(* CODESYS project rscommcommon.library
   Company: ESO
   Description: Common library for all rsComm projects.
   Version: 0.2.0.2
   Placeholder: ESO LDC Comm Common Library
   Title: ESO LDC Comm Common Library

Project tree, tasks and I/O mapping:
  libraries: Tc2_Standard, * (Beckhoff Automation GmbH); Tc2_System, * (Beckhoff Automation GmbH); Tc2_Utilities, * (Beckhoff Automation GmbH); Tc3_Module, * (Beckhoff Automation GmbH)
  DUTs/
    Enumerated/
      Comm/
        data type E_MODBUS_CMD_TYPE
        data type E_RS_BASE_READ_TYPE
        data type E_RS_COMM_CMD
        data type E_RS_COMM_ERROR
        data type E_RS_COMM_STATE
        data type E_RS_COMM_STATUS
        data type E_RS_COMMAND
        data type E_RS_RPC_ERROR
      Devices/
        data type E_LAKESHORE_CMD_TYPE
        data type E_LAKESHORE_ERROR
        data type E_RS_BASE_STATE
        data type E_RS_BASE_SUBSTATE
        data type E_SM_ERROR
        data type E_SM_EVENT
        data type E_SM_STATUS
    Structures/
      Comm/
        data type T_READING_LREAL
        data type T_RS_COMM_CFG
        data type T_RS_COMM_CTRL
        data type T_RS_COMM_INFO
        data type T_RS_COMM_STAT
      Devices/
        data type T_LAKESHORE_CFG
        data type T_LAKESHORE_COMMAND
        data type T_LAKESHORE_CTRL
        data type T_LAKESHORE_INFO
        data type T_LAKESHORE_STAT
        data type T_RS_BASE_CFG
        data type T_RS_BASE_CTRL
        data type T_RS_BASE_STAT
  GVLs/
  lib/
  POUs/
    function block FB_LAKESHORE_BASE [ST]: ActionInitExecute, ActivityInitializing, ActivityMonitoring, ActivityMonitoringUser, CheckForEvents, M_CheckCmdIndex, M_Configure, M_GetCommand, M_GetCommInitialised, M_GetCommStatus, M_GetCouplerState, M_RampDisable, M_RampEnable, M_ReadFromReply, M_UpdateStatus, ProcessEvents
    function block FB_RS_BASE [ST]: ActionDisableExecute, ActionEnableExecute, ActionErrExecute, ActionInitExecute, ActionResetExecute, ActionStopExecute, ActionUnexpExecute, ActivityInitializing, ActivityMonitoring, ActivityMonitoringUser, CheckForEvents, M_Configure, M_GetCouplerState, M_GetRpcErrorText, M_ReadSensors, M_SetLastGoodSubstate, M_SetRpcStatus, ProcessEvents, RPC_Disable, RPC_Enable, RPC_Init, RPC_Reset, RPC_Stop, SetAction, SetEvent, SetLastCommand, SetState, SetStatus
    function block FB_SIM_MODBUS_COMM_BASE [ST]: M_ActivityDo, M_ByteSwap_INT_TO_BYTES, M_ByteSwap_INT_TO_STRING, M_ByteSwap_REAL_TO_BYTES, M_ByteSwap_REAL_TO_STRING, M_ByteSwap_UINT_TO_BYTES, M_ByteSwapINT, M_ByteSwapREAL, M_GenerateRandom_INT, M_GenerateRandom_REAL, M_GetSimReply, M_InsertBytes_INT, M_InsertBytes_REAL
    function block FB_SIM_MODBUS_COMM_JUMO [ST]: M_GetSimReply
    function block FB_SIM_RS_COMM_BASE [ST]: M_ActivityDo, M_GenerateRandom_LREAL, M_Get_INT_TO_STRING, M_Get_LREAL_TO_STRING, M_GetRandom_LREAL_TO_STRING, M_GetSimReply
    function block FB_SIM_RS_COMM_DUMMY [ST]: M_ActivityDo, M_GetSimReply
    function block FB_SIM_RS_COMM_LAKESHORE [ST]: M_ActivityDo, M_GetSimReply
    program MAIN [ST]
  VISUs/
*)

// DUTs/Enumerated/Comm/E_MODBUS_CMD_TYPE
{attribute 'qualified_only'}
{attribute 'strict'}
TYPE E_MODBUS_CMD_TYPE :
(
	READ	:=	0,
	WRITE	:=	1
);
END_TYPE

// DUTs/Enumerated/Comm/E_RS_BASE_READ_TYPE
{attribute 'qualified_only'}
{attribute 'strict'}
TYPE E_RS_BASE_READ_TYPE :
(
	SINGLE			:= 0,
	SINGLE_USER,
	PERIODIC,
	PERIODIC_USER
);
END_TYPE

// DUTs/Enumerated/Comm/E_RS_COMM_CMD
{attribute 'qualified_only'}
////{xxxattribute 'strict'}
TYPE E_RS_COMM_CMD :
(
	NONE		:=	0,
	INIT		:=	1,
	SEND		:=	2,
	DISCONNECT	:=	3
);
END_TYPE

// DUTs/Enumerated/Comm/E_RS_COMM_ERROR
{attribute 'qualified_only'}
//{attribute 'strict'}
TYPE E_RS_COMM_ERROR :
(
	OK				:= 0,
	NOT_IN_OP_STATE,
	NOT_INIT,
	TIMEOUT,
	LISTEN,
	ACCEPT,
	SEND,
	RECEIVE,
	WRONG_STATE,
	NOT_IDLE,
	CONNECT,
	DISCONNECT
);
END_TYPE

// DUTs/Enumerated/Comm/E_RS_COMM_STATE
{attribute 'qualified_only'}
{attribute 'strict'}
TYPE E_RS_COMM_STATE :
(
	NOT_INIT			:= 0,
	IDLE				:= 1,
	CONNECT				:= 2,
	RESET				:= 3,
	PREPARE_SEND		:= 5,
	SEND				:= 10,
	RECEIVE				:= 15,
	WAIT				:= 20,
	CLEAR_BUFFER		:= 40,
	WAIT_AFTER_SEND		:= 55,
	DISCONNECT			:= 60,

	ERROR				:= 100
);
END_TYPE

// DUTs/Enumerated/Comm/E_RS_COMM_STATUS
{attribute 'qualified_only'}
////{xxxattribute 'strict'}
TYPE E_RS_COMM_STATUS :
(
	NOT_INIT	:= -1,
	IDLE		:= 0,
	BUSY		:= 1,
	ERROR		:= 2
);
END_TYPE

// DUTs/Enumerated/Comm/E_RS_COMMAND
{attribute 'qualified_only'}
{attribute 'strict'}
TYPE E_RS_COMMAND :
(
	NONE	:= 0,
	
	RESET,
	INIT,
	STOP,
	ENABLE,
	DISABLE,
	
	READ,
	READ_USER,
	MONITOR,
	MONITOR_USER,
	STOPMON,
	
	CTRL_CMD
	
);
END_TYPE

// DUTs/Enumerated/Comm/E_RS_RPC_ERROR
{attribute 'qualified_only'}
//{attribute 'strict'}
TYPE E_RS_RPC_ERROR :
(
	OK					:= 0,
	NOT_OP				:= -1,			
	NOT_NOTOP_READY		:= -2,			
	NOT_NOTOP_NOTREADY	:= -3,			
	LOCAL				:= -4			
);
END_TYPE

// DUTs/Enumerated/Devices/E_LAKESHORE_CMD_TYPE
{attribute 'qualified_only'}
{attribute 'strict'}
TYPE E_LAKESHORE_CMD_TYPE :
(
	INIT := 0,
	READ,
	CTRL
);
END_TYPE

// DUTs/Enumerated/Devices/E_LAKESHORE_ERROR
TYPE E_LAKESHORE_ERROR :
(
	OK				:= 16#0000,
	NOT_IN_OP_STATE	:= 16#0001,
	NOT_INIT		:= 16#0002,
	TIMEOUT			:= 16#0004,
	COMM			:= 16#0008,
	WRONG_STATE		:= 16#0010,
	NOT_IDLE		:= 16#0020
);
END_TYPE

// DUTs/Enumerated/Devices/E_RS_BASE_STATE
{attribute 'qualified_only'}
//{attribute 'strict'}
TYPE E_RS_BASE_STATE :
(
	NONE	:= 0,
	NOTOP,
	OP
);
END_TYPE

// DUTs/Enumerated/Devices/E_RS_BASE_SUBSTATE
// Substates MUST match definitions in the WS driver that can be found in
// ICS/ifw/fcf/devmgr/devices/src/include/devmgr/devices/sensorConfig.hpp
// Never change them without consulting the team.
{attribute 'qualified_only'}
//{attribute 'strict'}
TYPE E_RS_BASE_SUBSTATE :
(
	NONE				:= 0,
	
	NOTOP_NOTREADY		:= 100,
	NOTOP_READY			:= 101,
	NOTOP_INITIALIZING	:= 102,
	NOTOP_ERROR			:= 199,
	
	OP_MONITORING   	:= 200,
	OP_IDLE         	:= 201,
	OP_MONITORING_USER	:= 202,
	OP_ERROR         	:= 299
);
END_TYPE

// DUTs/Enumerated/Devices/E_SM_ERROR
{attribute 'qualified_only'}
//{attribute 'strict'}
TYPE E_SM_ERROR :
(
	OK					:= 0,
	HW_NOT_OP,			
	WRONG_CMD,			
	INIT_FAILURE,		

	NOT_INITIALISED		:= 90,
	ZERO_POINTER		:= 100	// Simulator error
);
END_TYPE

// DUTs/Enumerated/Devices/E_SM_EVENT
TYPE E_SM_EVENT :
(
	NONE	:= 0,
	
	(* events corresponding to commands *)
	RESET,
	INIT,
	STOP,
	ENABLE,
	DISABLE,
	
	READ,
	READ_USER,
	MONITOR,
	MONITOR_USER,
	STOPMON,
	CTRL_CMD,
	
	(* 
		Events corresponding to internal events 
	*)
	INITDONE,
	READDONE,
	
	
	(* events mapped to HW signals *)
	HWOK,
	COMMOK,
	ERRCOMM,
	ERRHW,
	ERRINIT
	
);
END_TYPE

// DUTs/Enumerated/Devices/E_SM_STATUS
TYPE E_SM_STATUS :
(
	OK		:= 0,
	ERROR
);
END_TYPE

// DUTs/Structures/Comm/T_READING_LREAL
TYPE T_READING_LREAL :
STRUCT
	lrValue:	LREAL; 	// LREAL (DOUBLE)
END_STRUCT
END_TYPE

// DUTs/Structures/Comm/T_RS_COMM_CFG
TYPE T_RS_COMM_CFG :
STRUCT

	sCmdSuffix:		STRING(16) := '$0D$0A';	(* Terminator for command *)
	sReplySuffix:	STRING(16) := '$0D$0A';	(* Terminator for reply *)

	nTimeout:		DINT := 3000;			(* Timeout on command reply. ALWAYS use ms for time !!! *)

END_STRUCT
END_TYPE

// DUTs/Structures/Comm/T_RS_COMM_CTRL
TYPE T_RS_COMM_CTRL :
STRUCT
	(* CTRL *)
	nCommand:		E_RS_COMM_CMD := E_RS_COMM_CMD.NONE;	(* Command Number, e.g. to INIT or SEND a command *)
	bExecute:		BOOL;						(* Setting to TRUE activates command *)

	sCmd:			STRING := '';				(* Command to be sent, e.g. '*IDN?' to get Lakeshore ID*)

	bHasReply:		BOOL;						(* If TRUE, there is a reply to the command *)

	nNumReplies:	DINT := 1;	(* Number of replies, i.e. number of cfg.sReplySuffix strings expected in the reply *)

END_STRUCT
END_TYPE

// DUTs/Structures/Comm/T_RS_COMM_INFO
TYPE T_RS_COMM_INFO :
STRUCT
(*
	Driver Information

	Change LOG:
	0.1 2018-02-07	- Copy of VLT RS_Comm_TC3 project @306329.
*)

	sDate:			STRING(32)	:= '2018-02-06';
	sDescription:	STRING(80) 	:= 'Serial Port Communication Drivers';
	sName:			STRING(64)	:= 'FB_RS_COMM';
	sPlatform:		STRING(32)	:= 'CoDeSys';
	sSynopsis:		STRING(64)	:= 'Serial Port Communication Drivers';
	nVersionMajor:	DINT		:= 0;
	nVersionMinor:	DINT		:= 1;


END_STRUCT
END_TYPE

// DUTs/Structures/Comm/T_RS_COMM_STAT
TYPE T_RS_COMM_STAT :
STRUCT
	(* STAT *)
	bInitialised:		BOOL := FALSE;		(* Flag if device is initialised *)
	bSimulation:		BOOL := FALSE;		(* Device simulated *)
	bConnected:			BOOL := FALSE;		(* Established connection status *)


	nLastCommand:		E_RS_COMM_CMD 		:= E_RS_COMM_CMD.NONE;
	nErrorCode:			E_RS_COMM_ERROR 	:= E_RS_COMM_ERROR.OK;
	nStatus: 			E_RS_COMM_STATUS	:= E_RS_COMM_STATUS.NOT_INIT; (* See E_RS_COMM_STATUS definitions *)

	sErrorText: 		STRING 	:= 'OK';
	sStatus:			STRING	:= '';			(* Status description *)

	sReply:				STRING(255);			(* Last  Reply from the device *)

END_STRUCT
END_TYPE

// DUTs/Structures/Devices/T_LAKESHORE_CFG
TYPE T_LAKESHORE_CFG EXTENDS T_RS_BASE_CFG:
STRUCT
	cmdList_Init:	ARRAY [1..8]	OF T_LAKESHORE_COMMAND;	// List of INIT commands
	cmdList_Read:	ARRAY [1..16] 	OF T_LAKESHORE_COMMAND;	// List of READ commands

	nModel:			DINT := 336;		// Supported models: 218, 224, 340 and 336.

END_STRUCT
END_TYPE

// DUTs/Structures/Devices/T_LAKESHORE_COMMAND
TYPE T_LAKESHORE_COMMAND :
STRUCT
	cmd:		STRING := '';	(* Command to send *)
	nReplies:	DINT;   		(* Number of replies, i.e. reply terminators *)
	nValues:	DINT;   		(* Number of returned numbers (values) in the reply *)
	offset:		DINT;			(* Offset in data array where to write the first value *)
END_STRUCT
END_TYPE

// DUTs/Structures/Devices/T_LAKESHORE_CTRL
TYPE T_LAKESHORE_CTRL EXTENDS T_RS_BASE_CTRL:
STRUCT
	sCmdUser:	T_LAKESHORE_COMMAND := (cmd := '*IDN?', nReplies := 1, nValues := 1, offset := 0);

	cmdList_Ctrl:	ARRAY [1..8] OF T_LAKESHORE_COMMAND;	// List of up to 8 Ctrl Commands (no '?')

	
	nPID_A_P:			UINT;		// P controller value
	nPID_A_I:			UINT;		// I controller value
	nPID_A_D:			UINT;		// D controller value
	nHeaterRange:		UINT;		// Resistance power range
	lrCtrlRamp:			LREAL;		// Delta-T Kelvin per minutes
	lrSetpoint_A:		LREAL;		// Setpoint [K]

END_STRUCT
END_TYPE

// DUTs/Structures/Devices/T_LAKESHORE_INFO
TYPE T_LAKESHORE_INFO :
STRUCT
(*
	Driver Information

	Change LOG:
	1.0	12/02/2014	- Ported from TC2.
	1.1	13/02/2014	- Addition of input parameters for Model and readout period.
	1.2	18/02/2014	- STATUS_LAKESHORE_ERROR := 1, to match IODev ICD.
					- Disabled OPC UA for comm instance of FB_RS_COMM.
	1.3 15/10/2014	- References Newest version always
					- Removed Tc2_OpcUa from References
	2.0 2016-08-10	- OPC UA notation with TMC Files
*)
	sDate:			STRING(16)	:= '2016-08-10';
	sDescription:	STRING(32) 	:= 'Lakeshore controller';
	sName:			STRING(16)	:= 'FB_LAKESHORE';
	sPlatform:		STRING(16)	:= 'CoDeSys';
	sSynopsis:		STRING(48)	:= 'EtherCAT PLC Lakeshore controller';
	nVersionMajor:	DINT		:= 2;
	nVersionMinor:	DINT		:= 0;

END_STRUCT
END_TYPE

// DUTs/Structures/Devices/T_LAKESHORE_STAT
TYPE T_LAKESHORE_STAT EXTENDS T_RS_BASE_STAT:
STRUCT

	nRetries:			UDINT := 0;			// Total number of retries in case of communication problems
	
	lrArrReadings:		ARRAY [0..31] OF	T_READING_LREAL;	// Array of readings

	sReply:				STRING(255); 		(* Last Lakeshore Reply to predefined commands*)
	sReplyUser:			STRING(255); 		(* Last Lakeshore Reply to USER command *)

	// Lakeshore readings
	lrKRDG_A:		LREAL;	// Temperature A [K]
	lrKRDG_B:		LREAL;	// Temperature B [K]
	lrCRDG_A:		LREAL;	// Temperature A [C]
	lrCRDG_B:		LREAL;	// Temperature B [C]

	nPID_P:			UINT;	// PID parameter P
	nPID_I:			UINT;	// PID parameter I
	nPID_D:			UINT;	// PID parameter D
	bRAMP_On:		BOOL;	// RAMP 1 On/Off state
	lrRAMP_Rate:	LREAL;	// RAMP rate
	lrSETP:			LREAL;	// Actual Setpoint [K]
	lrSETP_Target:	LREAL;	// Target Setpoint [K]
	lrHTR:			LREAL;	// Heater output [%]
	nRANGE:			UINT;	// Heater range

	nPID2_P:		UINT;	// PID2 parameter P
	nPID2_I:		UINT;	// PID2 parameter I
	nPID2_D:		UINT;	// PID2 parameter D
	bRAMP2_On:		BOOL;	// RAMP 2 On/Off state
	lrRAMP2_Rate:	LREAL;	// RAMP rate
	lrSETP2:		LREAL;	// Actual Setpoint 2 [K]
	lrSETP2_Target:	LREAL;	// Target Setpoint 2 [K]
	lrHTR2:			LREAL;	// Heater2 output [%]
	nRANGE2:		UINT;	// Heater2 range

	lrAOUT1:		LREAL;	// Analog Output 1
	lrAOUT2:		LREAL;	// Analog Output 2
	lrAOUT3:		LREAL;	// Analog Output 3
	lrAOUT4:		LREAL;	// Analog Output 4
	
	
END_STRUCT
END_TYPE

// DUTs/Structures/Devices/T_RS_BASE_CFG
TYPE T_RS_BASE_CFG :
STRUCT
	tDelay_Periodic:	TIME := T#5000MS;	// Delay between sets of PERIODIC reads.
	tDelay_Init:		TIME := T#500MS;	// Delay between INIT commands
	tDelay_Ctrl:		TIME := T#100MS;	// Delay between CTRL commands
	bAutoMonitor:		BOOL := TRUE;		// If true, it starts PERIODIC reads (monitoring) after INIT
END_STRUCT
END_TYPE

// DUTs/Structures/Devices/T_RS_BASE_CTRL
TYPE T_RS_BASE_CTRL :
STRUCT
	(* CTRL *)
// DPO	nCommand:	E_RS_COMM_CMD := E_RS_COMM_CMD.NONE;
	nCommand:	E_RS_COMMAND := E_RS_COMMAND.NONE;
	bExecute:	BOOL;
	
	// User parameters used with E_RS_COMMAND.CTRL_CMD,
	// when device specific commands have to be defined.
	// Command can be specified with a combination of parameters.
	// For example:
	//    cmd := E_RS_COMMAND.CTRL_CMD & nPar1 := 1  ==> cmd = 'start pulse'
	//    cmd := E_RS_COMMAND.CTRL_CMD & nPar1 := 2  ==> cmd = 'stop pulse'
	//    cmd := E_RS_COMMAND.CTRL_CMD & nPar1 := 3  ==> cmd = 'reload'
	nPar1:		DINT;
	nPar2:		DINT;
	nPar3:		DINT;
	
	lrPar1:		LREAL;
	lrPar2:		LREAL;
	lrPar3:		LREAL;
END_STRUCT
END_TYPE

// DUTs/Structures/Devices/T_RS_BASE_STAT
TYPE T_RS_BASE_STAT :
STRUCT
	bInitialised:	BOOL 	:= FALSE;		// Flag if device is initialised
	bConfigured:	BOOL 	:= FALSE;		// Flag if device is configured
	bLocal:			BOOL	:= FALSE;		// Device operated from PLC GUI
	bSimulation:	BOOL	:= FALSE;		// Device simulated
	bAutoStarted:	BOOL	:= FALSE;		// Device has already automatically got to OP state
	bActive:		BOOL	:= FALSE;		// Device has passed first 100 cycles
	bCmdActive:		BOOL 	:= FALSE;		// Flag if there are SET commands to be executed.
	bWaitUpdate:	BOOL 	:= FALSE;		// Flag if system waits for the update of status.
	bStatUpdated:	BOOL 	:= FALSE;		// Flag if status has been updated after SET commands.

	nState:			E_RS_BASE_STATE		:= E_RS_BASE_STATE.NOTOP;			
	nSubstate:		E_RS_BASE_SUBSTATE	:= E_RS_BASE_SUBSTATE.NOTOP_NOTREADY;

	nCycleCounter:	UDINT	:= 0;							// Alive flag
	nErrorCode: 	E_SM_ERROR 		:= E_SM_ERROR.OK;		(* Error code *)
	nLastCommand:	E_RS_COMMAND	:= E_RS_COMMAND.NONE;	(* Last command sent to the device *)
	nStatus: 		E_SM_STATUS		:= E_SM_STATUS.OK; 		(* Device status *)
	nRpcErrorCode: 	E_RS_RPC_ERROR 	:= E_RS_RPC_ERROR.OK;	(* RPC Error code *)

	sState:			STRING	:= 'NOT OP';					(* State textual description *)
	sSubstate:		STRING	:= 'NOT READY';					(* Substate textual description *)
	sErrorText: 	STRING 	:= 'OK'; 						(* Error text *)
	sRpcErrorText: 	STRING 	:= 'OK'; 						(* RPC Error text *)
	sStatus: 		STRING 	:= 'OK'; 						(* Status in textual form, e.g. 'OFF' *)
	sLastCommand:	STRING	:= 'NONE';						(* Last command, as string, sent to the device *)
	
	sActionDesc:	STRING	:= '';
	sEventDesc:		STRING	:= '';
END_STRUCT
END_TYPE

// POUs/FB_LAKESHORE_BASE
FUNCTION_BLOCK FB_LAKESHORE_BASE EXTENDS FB_RS_BASE
VAR_INPUT
	{attribute 'OPC.UA.DA' := '0'}
	in_nModel:			DINT := 340;	// Supported models: 218, 224, 336 and 340, default 340
	{attribute 'OPC.UA.DA' := '0'}
	in_bAutoMonitor:	BOOL := TRUE;	// If true, it starts PERIODIC reads (monitoring) after INIT
	{attribute 'OPC.UA.DA' := '0'}
	in_nPeriod:		DINT := 10000;		// Interval for periodic reading [ms], default 10000 ms = 10 sec
	{attribute 'OPC.UA.DA' := '0'}
	in_sCmdSuffix:		STRING(16);		// Terminator for command: LS336 '$0A', LS224 '$0D$0A'
	{attribute 'OPC.UA.DA' := '0'}
	in_sReplySuffix:	STRING(16);		// Terminator for reply
END_VAR
VAR_OUTPUT
END_VAR
VAR CONSTANT
END_VAR
VAR
	{attribute 'OPC.UA.DA' := '1'}
	cfg:		T_LAKESHORE_CFG;	
	{attribute 'OPC.UA.DA' := '1'}
	ctrl:		T_LAKESHORE_CTRL;	
	{attribute 'OPC.UA.DA' := '1'}
	{attribute 'OPC.UA.DA.Access' := '1'}
	info:		T_LAKESHORE_INFO;	(* ReadOnly *)

	{attribute 'OPC.UA.DA' := '1'}
	{attribute 'OPC.UA.DA.Access' := '1'}
	stat:		T_LAKESHORE_STAT;	(* Common State Machine Status - ReadOnly *)

	
	// There are different configurations for each Lakeshore model.
	// That's why we need pointers, e.g. ptrReadCmds.
	// We also need pointers to structures inside FB_RS_COMM, e.g. ptrCommCfg.
	{attribute 'OPC.UA.DA' := '0'}
	ptrCommCfg:		POINTER TO T_RS_COMM_CFG;	(* Pointer to comm.cfg instance *)
	{attribute 'OPC.UA.DA' := '0'}
	ptrCommCtrl:	POINTER TO T_RS_COMM_CTRL;	(* Pointer to comm.ctrl instance *)
	{attribute 'OPC.UA.DA' := '0'}
	ptrCommStat:	POINTER TO T_RS_COMM_STAT;	(* Pointer to comm.stat instance *)


	(* Timers *)
	{attribute 'OPC.UA.DA' := '0'}
	fbTimer:		TON; (* General Timeout *)

	(* Misc internal vars *)
	{attribute 'OPC.UA.DA' := '0'}
	cmdCounter:		INT := 1;	// Position in commands table
	{attribute 'OPC.UA.DA' := '0'}
	bResult:		BOOL := FALSE;
END_VAR

// Set references
cfgRef	REF=cfg;
ctrlRef	REF=ctrl;
statRef	REF=stat;


// Execute the base class object FB_RS_BASE
SUPER^();

METHOD ActionInitExecute
VAR_INPUT
END_VAR
// Populate cfg.cmdList_Init and cmdList_Read tables for the specific cfg.nModel.
M_Configure();

SUPER^.ActionInitExecute();
END_METHOD

METHOD ActivityInitializing
VAR_INPUT
	bExecute:	BOOL;
END_VAR
VAR_INST
	{attribute 'OPC.UA.DA' := '0'}
    nMethodState:	INT := 0;	// State Machine current state
END_VAR
SetAction('ActivityInitializing');


IF NOT bExecute THEN
	nMethodState	:= 0;	// Reset the state machine
	cmdCounter		:= 0;	// Start from the first init command (after increment in state 15)
	RETURN;
END_IF

// Handle State Machine
CASE nMethodState OF
	0:	
		(* Set initial state and status *)
		stat.bInitialised	:= FALSE;
		stat.sReply			:= '';
		SetStatus(E_SM_ERROR.OK, 'BUSY');

		nMethodState := 10;				// Go to next state, i.e. INIT_COMM

	10:	// Initialize COMM port
		(* Reset the serial port *)
		ptrCommCtrl^.nCommand	:= E_RS_COMM_CMD.INIT;
		ptrCommCtrl^.bExecute	:= TRUE;

		(* Start the timer by going false/true *)
		fbTimer (IN := FALSE); (* Reset timer *)
		fbTimer (IN := TRUE, PT := T#5S); (* 5 sec timeout for reply *)

		nMethodState 	:= 15;	// On next cycle wait until the comm port is reset, i.e. idle
		
	15:	// Wait IDLE
		fbTimer (IN := TRUE);
		IF M_GetCommStatus() = E_RS_COMM_STATUS.IDLE  AND M_GetCommInitialised() THEN
			// Communication is IDLE 
			fbTimer (IN := FALSE);	// disable timer 
			stat.sReply		:= ptrCommStat^.sReply;	// Save the reply
			cmdCounter		:= cmdCounter + 1;	// Increment init command index
			fbTimer (IN := FALSE);	// disable timer 
			fbTimer (IN := TRUE, PT := cfg.tDelay_Init); // Wait INIT delay
			bCommProblem	:= FALSE;
			nMethodState 	:= 18;	// Execute next device INIT command
		ELSIF M_GetCommStatus() = E_RS_COMM_STATUS.ERROR THEN
			fbTimer (IN := FALSE);
			SetStatus(E_LAKESHORE_ERROR.COMM, 'ERROR: Communication error');	
			bCommProblem	:= TRUE;
			nEvent := E_SM_EVENT.ERRINIT;
			RETURN;
		ELSIF fbTimer.Q THEN
			// Timer expired after 5 sec. This is an error.
			fbTimer (IN := FALSE);
			SetStatus(E_LAKESHORE_ERROR.TIMEOUT, 'ERROR: Communication timeout');	
			bCommProblem	:= TRUE;
			nEvent := E_SM_EVENT.ERRINIT;
			RETURN;
		END_IF

	
	
	18:	// Wait INIT Delay
		fbTimer (IN := TRUE);
		IF fbTimer.Q THEN
			// Timer expired after 5 sec. This is an error.
			fbTimer (IN := FALSE);
			nMethodState 	:= 20;	// Execute next device INIT command
			RETURN;
		END_IF

	
	
	20:	// INIT DEV
//		IF ptrInitCmds^ [cmdCounter].cmd = '' THEN
		IF cfg.cmdList_Init[cmdCounter].cmd = '' THEN
			// Device INIT is done. Go to IDLE 
			stat.bInitialised 	:= TRUE;
			cmdCounter			:= 1;
			SetStatus(E_SM_ERROR.OK, 'IDLE');
			nEvent 		:= E_SM_EVENT.INITDONE;
			RETURN;
		END_IF
		
		(* Send INIT command with index cmdCounter *)
		ptrCommCtrl^.nCommand		:= E_RS_COMM_CMD.SEND;
		ptrCommCtrl^.sCmd			:= cfg.cmdList_Init[cmdCounter].cmd;
		ptrCommCtrl^.nNumReplies	:= cfg.cmdList_Init[cmdCounter].nReplies;
		ptrCommCtrl^.bHasReply		:= cfg.cmdList_Init[cmdCounter].nReplies > 0;
		ptrCommCtrl^.bExecute		:= TRUE;
	
		(* Start the timer by going false/true *)
		fbTimer (IN := FALSE); (* Reset timer *)
		fbTimer (IN := TRUE, PT := T#5S); (* 5 sec timeout for reply *)

		// On next cycle wait until the comm port is idle
		nMethodState 	:= 15;	// On next cycle wait until the comm port is idle
	
END_CASE
END_METHOD

METHOD ActivityMonitoring
VAR_INPUT
	bExecute:	BOOL;
END_VAR
VAR
END_VAR
VAR_INST
	{attribute 'OPC.UA.DA' := '0'}
    nMethodState:	INT := 0;	// State Machine current state
	{attribute 'OPC.UA.DA' := '0'}
	nRetries:		INT := 0;	// Number of retries in case of communication problems
	{attribute 'OPC.UA.DA' := '0'}
	nCmdType:		E_LAKESHORE_CMD_TYPE := E_LAKESHORE_CMD_TYPE.READ;
	{attribute 'OPC.UA.DA' := '0'}
	devCmd:			T_LAKESHORE_COMMAND;	// Device command to be sent
END_VAR
IF NOT cfg.bAutoMonitor AND stat.nSubstate = E_RS_BASE_SUBSTATE.NOTOP_READY THEN
	SetAction('No Monitoring'); 
	SetStatus(E_SM_ERROR.OK, 'IDLE');
	nMethodState	:= 0;	// Reset the state machine
	cmdCounter		:= 1;	// Reading will start from the first command in the array
	RETURN;
END_IF

IF NOT bExecute THEN
	SetAction('ActivityMonitoring'); 
	SetStatus(E_SM_ERROR.OK, 'BUSY');
	nMethodState	:= 0;	// Reset the state machine
	nCmdType		:= E_LAKESHORE_CMD_TYPE.READ;	// We start with READ commands.
	cmdCounter		:= 1;	// Reading will start from the first command in the array
	RETURN;
END_IF

// Handle State Machine
CASE nMethodState OF
	0:	// Execute a command from the command array.
		// Note that command might be READ or CTRL type (see nCmdType)!
		devCmd	:= M_GetCommand(nCmdType, cmdCounter);	// Get command
		IF nCmdType = E_LAKESHORE_CMD_TYPE.READ  AND devCmd.cmd = '' THEN
			// We have executed all READ commands.
			// Update status, i.e. copy readings from stat.lrArrReadings[] to dedicated variables.
			M_UpdateStatus();
			
			// If this is the first round of READ commands after the CTRL commands,
			// Indicate it with the stat.bStatUpdated flag.
			// This means that the CTRL commands have been executed and the status
			// was updated after that.
			IF stat.bWaitUpdate	THEN
				stat.bWaitUpdate	:= FALSE;
				stat.bStatUpdated	:= TRUE;
			END_IF
			
			// We arrived to the end of the array of pre-defined READ commands.
			// Check if we have to exit Monitoring
			IF nNextState <> E_RS_BASE_STATE.NONE	THEN
				SetStatus(E_SM_ERROR.OK, nNextDescription);
				SetState(nNextState, nNextSubstate);
				nNextState		:= E_RS_BASE_STATE.NONE;
				nNextSubstate	:= E_RS_BASE_SUBSTATE.NONE;
				nNextDescription:= '';
				RETURN;
			ELSIF nReadType = E_RS_BASE_READ_TYPE.SINGLE	THEN
				// If it's a single read, exit here.
				SetStatus(E_SM_ERROR.OK, 'IDLE');
				nInternalEvent := E_SM_EVENT.READDONE;
				RETURN;
			END_IF

			// Periodic READ is done. 
			// We set the counter back to one. 
			cmdCounter	:= 1;
			
			// Check if there are some CTRL commands to be executed as well.
			IF stat.bCmdActive THEN
				// Switch to CTRL commands.
				nCmdType	:= E_LAKESHORE_CMD_TYPE.CTRL;
				devCmd		:= M_GetCommand(nCmdType, cmdCounter);	// Get command
			ELSE
				// Wait tDelay_Periodic before re-starting the READ.
				SetStatus(E_SM_ERROR.OK, 'IDLE');
				
				(* Start the timer by going false/true *)
				fbTimer (IN := FALSE); (* Reset timer *)
				fbTimer (IN := TRUE, PT := cfg.tDelay_Periodic);
				cmdCounter		:= 1;	// Reading will start from the first command in the array
				nMethodState 	:= 10;	// Goto Wait for tDelay_Periodic
				RETURN;
			END_IF
		ELSIF nCmdType = E_LAKESHORE_CMD_TYPE.CTRL  AND devCmd.cmd = '' THEN
			// We have executed all CTRL commands.
			// Indicate it by setting stat.bWaitUpdate, i.e.
			// we will wait for another round of READ commands in order
			// to update the status after CTRL commands.
			// After that, stat.bStatUpdated will be set to TRUE.
			stat.bCmdActive		:= FALSE;
			stat.bWaitUpdate	:= TRUE;
			stat.bStatUpdated	:= FALSE;
			
			// We set the counter back to one. 
			cmdCounter	:= 1;
			// Next round will start with Periodic READ. 
			nCmdType	:= E_LAKESHORE_CMD_TYPE.READ;
			
			// Wait tDelay_Periodic before re-starting the READ.
			SetStatus(E_SM_ERROR.OK, 'IDLE');
			
			(* Start the timer by going false/true *)
			fbTimer (IN := FALSE); (* Reset timer *)
			fbTimer (IN := TRUE, PT := cfg.tDelay_Periodic);
			nMethodState := 10;				// Goto Wait for tDelay_Periodic
			RETURN;
		END_IF
		
		(* Send command with index cmdCounter *)
		ptrCommCtrl^.nCommand		:= E_RS_COMM_CMD.SEND;
		ptrCommCtrl^.sCmd			:= devCmd.cmd;
		ptrCommCtrl^.nNumReplies	:= devCmd.nReplies;
		ptrCommCtrl^.bHasReply		:= devCmd.nReplies > 0;
		ptrCommCtrl^.bExecute		:= TRUE;

		statRef.sErrorText	:= 'BUSY';

		// In case we are executing a CTRL commands, there are no replies.
		// However, we apply a delay tDelay_Ctrl that is at least 50ms.
		IF NOT ptrCommCtrl^.bHasReply THEN
			fbTimer (IN := FALSE); // Reset timer
			fbTimer (IN := TRUE, PT := cfgRef.tDelay_Ctrl); 
			cmdCounter		:= cmdCounter + 1;	// Go to next command.
			nMethodState	:= 10;				// Goto WAIT for delay
			RETURN;
		ELSE			
			// There is a reply, i.e. this is a 'READ' command.
			// Apply short delay of 10ms before checking the status of comm port. 
			// Start the timer by going false/true
			fbTimer (IN := FALSE); // Reset timer
			fbTimer (IN := TRUE, PT := T#10MS);	
			statRef.sErrorText	:= 'BUSY';
			nMethodState := 15;	// Goto short delay
		END_IF
		
		
		
	10:	// Wait until the delay timeout expires
		fbTimer (IN := TRUE);

		// Check if we have to exit Monitoring
		IF nNextState <> E_RS_BASE_STATE.NONE THEN
			fbTimer (IN := FALSE); (* Stop the timer *)
			SetStatus(E_SM_ERROR.OK, nNextDescription);
			SetState(nNextState, nNextSubstate);
			nNextState		:= E_RS_BASE_STATE.NONE;
			nNextSubstate	:= E_RS_BASE_SUBSTATE.NONE;
			nNextDescription:= '';
			RETURN;
		END_IF
	
		(* If Timer has expired, go to the next state. *)
		IF fbTimer.Q THEN
			fbTimer (IN := FALSE);
			nMethodState 	:= 0;				// Goto handling of next command
			RETURN;
		END_IF
	
	15:	// Wait until the delay timeout expires
		fbTimer (IN := TRUE);

		(* If Timer has expired, go to the next state. *)
		IF fbTimer.Q THEN
			fbTimer (IN := FALSE);
			fbTimer (IN := TRUE, PT := T#3S);	// 3 sec timeout for reply
			statRef.sErrorText	:= 'BUSY';
			nMethodState 	:= 20;	// Goto Wait for IDLE/Reply
			RETURN;
		END_IF
	



	20:	// Wait for the reading to complete, i.e. IDLE
		fbTimer (IN := TRUE);
		IF M_GetCommStatus() = E_RS_COMM_STATUS.IDLE THEN
			// Communication is IDLE 
			fbTimer (IN := FALSE);	// disable timer 
			stat.sReply		:= ptrCommStat^.sReply;	// Save the reply
			
			// Extract values from the reply.
			// The values are stored into stat.lrArrReadings array.
			M_ReadFromReply(idx := DINT_TO_INT(devCmd.offset),
							n 	:= DINT_TO_INT(devCmd.nValues),
							str := stat.sReply,
							ok 	=> bResult);

			bCommProblem	:= FALSE;
			nRetries		:= 0;	// Reset number of retries

			
			// Check if we have to exit Monitoring
			IF nNextState <> E_RS_BASE_STATE.NONE THEN
				fbTimer (IN := FALSE); (* Stop the timer *)
				SetStatus(E_SM_ERROR.OK, nNextDescription);
				SetState(nNextState, nNextSubstate);
				nNextState		:= E_RS_BASE_STATE.NONE;
				nNextSubstate	:= E_RS_BASE_SUBSTATE.NONE;
				nNextDescription:= '';
				RETURN;
			END_IF
	
			cmdCounter		:= cmdCounter + 1;	// Increment command index
			
			nMethodState 	:= 0;				// Goto Send command
			nEvent := E_SM_EVENT.COMMOK;
			RETURN;
		ELSIF M_GetCommStatus() = E_RS_COMM_STATUS.ERROR OR fbTimer.Q THEN
			fbTimer (IN := FALSE);
			SetStatus(E_LAKESHORE_ERROR.COMM, 'ERROR: Communication error');	
			bCommProblem	:= TRUE;
			// Retry up to 2 times
			nRetries		:= nRetries + 1;		// Increment number of retries
			stat.nRetries	:= stat.nRetries + 1;	// Increment total number of retries
			IF nRetries > 1 THEN
				nEvent := E_SM_EVENT.ERRCOMM;
				RETURN;
			END_IF
			// Apply a short delay of 1 sec and retry
			fbTimer (IN := FALSE); (* Reset timer *)
			fbTimer (IN := TRUE, PT := T#1000MS);
			nMethodState := 10;				// Goto Wait 
			RETURN;
		END_IF

	
END_CASE
END_METHOD

METHOD ActivityMonitoringUser
VAR_INPUT
	bExecute:	BOOL;
END_VAR
VAR_INST
	{attribute 'OPC.UA.DA' := '0'}
    nMethodState:	INT := 0;	// State Machine current state
	{attribute 'OPC.UA.DA' := '0'}
	nRetries:		INT := 0;	// Number of retries in case of communication problems
END_VAR

IF NOT bExecute THEN
	SetAction('ActivityMonitoringUser'); 
	SetStatus(E_SM_ERROR.OK, 'BUSY');
	nMethodState	:= 0;	// Reset the state machine
	RETURN;
END_IF

// Handle State Machine
CASE nMethodState OF
	0:	// Execute the User command ctrl.sCmdUser.cmd
		
		ptrCommCtrl^.nCommand		:= E_RS_COMM_CMD.SEND;
		ptrCommCtrl^.sCmd			:= ctrl.sCmdUser.cmd;
		ptrCommCtrl^.nNumReplies	:= ctrl.sCmdUser.nReplies;
		ptrCommCtrl^.bHasReply		:= ctrl.sCmdUser.nReplies > 0;
		ptrCommCtrl^.bExecute		:= TRUE;
		
		(* Start the timer by going false/true *)
		fbTimer (IN := FALSE); (* Reset timer *)
		fbTimer (IN := TRUE, PT := T#5S); (* 5 sec timeout for reply *)

		nMethodState := 20;				// Goto WAIT for Reading to complete,

	10:	// Wait until the delay timeout expires
		fbTimer (IN := TRUE);

		// Check if we have to exit Monitoring
		IF nNextState <> E_RS_BASE_STATE.NONE THEN
			fbTimer (IN := FALSE); (* Stop the timer *)
			SetStatus(E_SM_ERROR.OK, nNextDescription);
			SetState(nNextState, nNextSubstate);
			nNextState		:= E_RS_BASE_STATE.NONE;
			nNextSubstate	:= E_RS_BASE_SUBSTATE.NONE;
			nNextDescription:= '';
			RETURN;
		END_IF
	
		(* If Timer has expired, go to the next state. *)
		IF fbTimer.Q THEN
			fbTimer (IN := FALSE);
			SetStatus(E_SM_ERROR.OK, 'BUSY');
			nMethodState 	:= 0;				// Goto Wait for tDelay_Periodic
			RETURN;
		END_IF
	


	20:	// Wait for the reading to complete, i.e. IDLE
		fbTimer (IN := TRUE);
		IF M_GetCommStatus() = E_RS_COMM_STATUS.IDLE THEN
			// Communication is IDLE 
			fbTimer (IN := FALSE);	// disable timer 
			
			// Save the reply. That's all since we don't know how too process the reply
			stat.sReplyUser	:= ptrCommStat^.sReply;	
			
			bCommProblem	:= FALSE;
			nRetries		:= 0;	// Reset number of retries

			
			// Check if we have to exit Monitoring
			IF nNextState <> E_RS_BASE_STATE.NONE THEN
				fbTimer (IN := FALSE); (* Stop the timer *)
				SetStatus(E_SM_ERROR.OK, nNextDescription);
				SetState(nNextState, nNextSubstate);
				nNextState		:= E_RS_BASE_STATE.NONE;
				nNextSubstate	:= E_RS_BASE_SUBSTATE.NONE;
				nNextDescription:= '';
				RETURN;
			ELSIF nReadType <> E_RS_BASE_READ_TYPE.PERIODIC_USER	THEN
				// This was single READ_USER
				SetStatus(E_SM_ERROR.OK, 'IDLE');
				nInternalEvent := E_SM_EVENT.READDONE;
				RETURN;
			ELSE
				// Periodic READ is done. Wait tDelay_Periodic before re-starting the READ.
				SetStatus(E_SM_ERROR.OK, 'IDLE');
				
				(* Start the timer by going false/true *)
				fbTimer (IN := FALSE); (* Reset timer *)
				fbTimer (IN := TRUE, PT := cfg.tDelay_Periodic);
				nMethodState := 10;				// Goto Wait for tDelay_Periodic
			END_IF
			RETURN;
		ELSIF M_GetCommStatus() = E_RS_COMM_STATUS.ERROR OR fbTimer.Q THEN
			fbTimer (IN := FALSE);
			SetStatus(E_LAKESHORE_ERROR.COMM, 'ERROR: Communication error');	
			bCommProblem	:= TRUE;
			// Retry up to 3 times
			nRetries		:= nRetries + 1;		// Increment number of retries
			stat.nRetries	:= stat.nRetries + 1;	// Increment total number of retries
			IF nRetries > 3 THEN
				nEvent := E_SM_EVENT.ERRCOMM;
			ELSE
				// Apply a short delay of 1 sec and retry
				fbTimer (IN := FALSE); (* Reset timer *)
				fbTimer (IN := TRUE, PT := T#1000MS);
				nMethodState := 10;				// Goto Wait 
			END_IF
			RETURN;
		END_IF

	
END_CASE
END_METHOD

METHOD CheckForEvents
VAR_INPUT
END_VAR
VAR
END_VAR

(* 
	Start assuming the HW is OK in case there was no communication problem. 
	This is needed to recover from the situation where 
	the HW was failing and now it is working.
*)

//IF NOT bCommProblem	THEN
//	nInternalEvent := E_SM_EVENT.HWOK;
//END_IF




(* 
	Check for events in the following order: 
   	1) HW failure: without HW avilability there is no point to do anything
	2) Internal events: to allow completing the initiated commands before 
                        starting processing new commands. 
   	3) Commands: to react to external commands. Commands should be executed 
                 before processing HW signals to allow to start a recovery action.
   	4) HW signals: if any.
*)

IF NOT M_GetCouplerState() THEN	
	(* Check if the HW is NOT OK *)
	(*
	If the hardware status is NOT OK, we cannot trust the readings.
	Variable i_nCouplerState has to be mapped to a State of a terminal, e.g. EK1100.
	The value should be 8.
 	*)
	SetEvent(E_SM_EVENT.ERRHW);
	SetStatus(E_SM_ERROR.HW_NOT_OP, 'ERROR: HW not in OPERATIONAL state');
	
ELSIF M_GetCouplerState() AND stat.nErrorCode = E_SM_ERROR.HW_NOT_OP THEN
	SetEvent(E_SM_EVENT.HWOK);

ELSIF ctrlRef.bExecute  THEN
	(* Handle commands *)
	ctrlRef.bExecute		:= FALSE;			(* Clear the Execute bit *)
	SetLastCommand(ctrlRef.nCommand);			(* Save the last command *)
	SetEvent(ctrlRef.nCommand);
	ctrlRef.nCommand 		:= E_RS_COMMAND.NONE;	(* Clear the Command *)
ELSIF nInternalEvent <> E_SM_EVENT.NONE THEN
	(* Handle internal events *)
	SetEvent(nInternalEvent);
	nInternalEvent := E_SM_EVENT.NONE;
ELSE
	(* Handle HW problems and unexpected bahaviour *)
	
END_IF
END_METHOD

METHOD M_CheckCmdIndex : BOOL
VAR_INPUT
	in_nCmdType:	E_LAKESHORE_CMD_TYPE;
	in_nIndex:		INT;
END_VAR
CASE in_nCmdType OF
	E_LAKESHORE_CMD_TYPE.INIT,
	E_LAKESHORE_CMD_TYPE.CTRL:
		// INIT and CTRL commands have index [1..8].
		// The index of the command must be between 1 and 8.
		IF in_nIndex < 1  OR  in_nIndex > 8 THEN
			M_CheckCmdIndex	:= FALSE;
		ELSE
			M_CheckCmdIndex	:= TRUE;
		END_IF
	E_LAKESHORE_CMD_TYPE.READ:
		// READ commands have index [1..16].
		// The index of the command must be between 1 and 16.
		IF in_nIndex < 1  OR  in_nIndex > 16 THEN
			M_CheckCmdIndex	:= FALSE;
		ELSE
			M_CheckCmdIndex	:= TRUE;
		END_IF
END_CASE
END_METHOD

METHOD M_Configure
VAR_INPUT
END_VAR
// Copy input parameters to configuration
cfg.nModel			:= in_nModel;
cfg.bAutoMonitor	:= in_bAutoMonitor;
cfg.tDelay_Periodic	:= DINT_TO_TIME(in_nPeriod);


// TODO in FB that extends the functionality
// Set pointers to comm, i.e.
//	ptrCommCfg	:= ADR(comm.cfg);		(* Pointer to comm.cfg instance *)
//	ptrCommCtrl	:= ADR(comm.ctrl);	(* Pointer to comm.ctrl instance *)
//	ptrCommStat	:= ADR(comm.stat);	(* Pointer to comm.stat instance *)
END_METHOD

METHOD M_GetCommand : T_LAKESHORE_COMMAND
VAR_INPUT
	in_nCmdType:	E_LAKESHORE_CMD_TYPE;
	in_nIndex:		INT;
END_VAR
VAR
	emptyCmd:	T_LAKESHORE_COMMAND;
END_VAR
IF NOT M_CheckCmdIndex(in_nCmdType, in_nIndex)	THEN
	// The index is not valid. Set empty command.
	M_GetCommand	:= emptyCmd;
	RETURN;
END_IF

CASE in_nCmdType OF
	E_LAKESHORE_CMD_TYPE.INIT:
		M_GetCommand	:= cfg.cmdList_Init  [in_nIndex];
	E_LAKESHORE_CMD_TYPE.READ:
		M_GetCommand	:= cfg.cmdList_Read  [in_nIndex];
	E_LAKESHORE_CMD_TYPE.CTRL:
		M_GetCommand	:= ctrl.cmdList_Ctrl [in_nIndex];
END_CASE
END_METHOD

METHOD M_GetCommInitialised : BOOL
VAR_INPUT
END_VAR
// TODO: In each extended FB add the following:
// M_GetCommInitialised	:= comm.M_GetInitialised();

// This is just a dummy method for BASE FB
M_GetCommInitialised	:= FALSE;
END_METHOD

METHOD M_GetCommStatus : E_RS_COMM_STATUS
VAR_INPUT
END_VAR
// TODO: In each extended FB add the following:
// M_GetCommStatus	:= comm.M_GetStatus();

// This is just a dummy method for BASE FB
M_GetCommStatus	:= E_RS_COMM_STATUS.ERROR;
END_METHOD

METHOD M_GetCouplerState : BOOL
VAR_INPUT
END_VAR
M_GetCouplerState	:= TRUE;
END_METHOD

METHOD M_RampDisable
VAR_INPUT
END_VAR
// Disable the RAMP by setting all parameters to zero and
// the SETP to the current temperature.
M_RampEnable(0, 0, 0, 0, 0, stat.lrKRDG_A);
END_METHOD

// Set Lakeshore PID and other control parameters
METHOD M_RampEnable
VAR_INPUT
	in_nPID_A_P:		UINT;		// P controler value
	in_nPID_A_I:		UINT;		// I controler value
	in_nPID_A_D:		UINT;		// D controler value
	in_nHeater_Range:	UINT;		// Resistance power range
	in_lrCtrlRamp:		LREAL;		// Delta-T Kelvin per minutes
	in_lrSetpoint_A:	LREAL;		// Setpoint [K]
END_VAR
VAR
	cmd:		STRING;
	fbFormat:	FB_FormatString;
	nRampOn:	UINT;
END_VAR
//
// This code will set PID parameters and start the ramp.
// However, in order to avoid big jump in the ramp, 
// the ramp should be disabled first and setpoint set to the current temperature.
// Then, target ramp and setpoint should be set again.
// That's why there is a double RAMP/SETP sequence.
//

// 'PID 1,50,71,10'
// 'RANGE 4'
// 'RAMP 1,0,0.0'
// 'SETP 1, <current temperature>', 
// 'RAMP 1,1,5.0'.
// 'SETP 1, <SET POINT>'.


//
//	Copy input parameters into ctrl parameters.
//
ctrl.nPID_A_P		:= in_nPID_A_P;
ctrl.nPID_A_I		:= in_nPID_A_I;
ctrl.nPID_A_D		:= in_nPID_A_D;
ctrl.nHeaterRange	:= in_nHeater_Range;
ctrl.lrCtrlRamp		:= in_lrCtrlRamp;
ctrl.lrSetpoint_A	:= in_lrSetpoint_A;

// Update SETP in status
stat.lrSETP_Target	:= ctrl.lrSetpoint_A;


//
//	Set command strings in ctrl.cmdList_Ctrl[].
//

//
// Set PID parameters, e.g. 'PID 1,50,71,10'.
// Index in ctrl.cmdList_Ctrl[] is 1
//
fbFormat(	sFormat := 'PID 1, %d, %d, %d', 
			arg1	:= F_UINT(ctrl.nPID_A_P), 
			arg2	:= F_UINT(ctrl.nPID_A_I), 
			arg3	:= F_UINT(ctrl.nPID_A_D), 
			sOut => cmd);
ctrl.cmdList_Ctrl[1].cmd	:= cmd;


//
// Set RANGE parameters, e.g. 'RANGE 4'.
// Index in ctrl.cmdList_Ctrl[] is 2
//
fbFormat(	sFormat := 'RANGE %d', 
			arg1 := F_UINT(ctrl.nHeaterRange), 
			sOut => cmd);
ctrl.cmdList_Ctrl[2].cmd	:= cmd;


//
// The following two command will set the SETP to the current Lakeshore temperature.
// This way ramping starts from the current temperature and not from
// the last SETP.
// In this trick, RAMP=0 & SETP=DET temperature.
// 'RAMP 1,0,0.0'  &  'SETP 1, <DET T>'
//
// Set RAMP to zero, i.e. 'RAMP 1,0,0.0'.
// Index in ctrl.cmdList_Ctrl[] is 3
//
ctrl.cmdList_Ctrl[3].cmd	:= 'RAMP 1,0,0.0';

//
// Set SETP to current DET temperature.
// Index in ctrl.cmdList_Ctrl[] is 4
//
fbFormat(	sFormat := 'SETP 1, %.2f', 
			arg1 := F_LREAL(stat.lrKRDG_A), 
			sOut => cmd);
ctrl.cmdList_Ctrl[4].cmd	:= cmd;


//
// Set RAMP parameters, e.g. 'RAMP 1,1,5.0'.
// Index in ctrl.cmdList_Ctrl[] is 5
// If ramp is zero, disable it.
//
nRampOn	:= BOOL_TO_UINT(ctrl.lrCtrlRamp > 0.0);
fbFormat(	sFormat := 'RAMP 1, %d, %.1f', 
			arg1	:= F_UINT(nRampOn),
			arg2	:= F_LREAL(ctrl.lrCtrlRamp), 
			sOut => cmd);
ctrl.cmdList_Ctrl[5].cmd	:= cmd;

//
// Set SETPOINT parameters, e.g. 'SETP 1,80.00'.
// Index in ctrl.cmdList_Ctrl[] is 6
//
fbFormat(	sFormat := 'SETP 1, %.2f', 
			arg1 := F_LREAL(ctrl.lrSetpoint_A), 
			sOut => cmd);
ctrl.cmdList_Ctrl[6].cmd	:= cmd;

//
// Flag the execution of CTRL commands.
// ActivityMonitoring() will see the flags and execute commands given in ctrl.cmdList_Ctrl[]
// after all monitoring (READ) commands given in cfg.cmdList_Read[] are completed.
// When everything is completed, stat.bStatUpdated will be set to TRUE.
// After that, new CTRL commands can be sent to the Lakeshore.
//
stat.bCmdActive		:= TRUE;	// This will switch from cmdList_Read to cmdList_Ctrl. 
stat.bWaitUpdate	:= FALSE;
stat.bStatUpdated	:= FALSE;
END_METHOD

METHOD M_ReadFromReply : BOOL
(* FB to extract 'n' values from 'str' and copy them into stat.lrArrReadings starting from index 'idx'.

	Example: 
		M_ReadFromReply (	idx := 5, 
							n := 3, 
							str := '0050.1,0020.2,0000$0D$0A', 
							ok => ok);
		res [5] = 50.1
		res [6] = 20.2
		res [7] = 0.0
		ok = TRUE
*)

VAR_INPUT
	idx:	INT;		(* arr [idx] will hold the first extracted value, arr [idx+1] the second one, etc. *)
	n:		INT;		(* Number of values to extract from the string - command specific *)
	str:	STRING(255);		(* String returned in Lakeshore reply *)
END_VAR
VAR_OUTPUT
	ok:		BOOL;		(* TRUE if the reading was correct, i.e. 'n' values successfully extracted from 'str'.  *)
END_VAR

VAR
	i:		INT;
	str_l:	STRING(255);
	pos:	INT;
END_VAR
i	:= 0;
str_l	:= str;
ok	:= TRUE; (* OK *)


WHILE i < n DO
	stat.lrArrReadings [idx + i].lrValue	:= STRING_TO_LREAL (str_l); (* take the first number *)
	(* move to just after the comma *)
	IF i < (n-1) THEN
		pos := FIND (str_l, ','); (* find the comma *)
		IF pos = 0 THEN (* less than 'n' numbers present in the string *)
			ok	:= FALSE; (* ERROR *)
			i 	:= n;
		ELSE
			str_l := RIGHT (str_l, LEN(str_l) - pos);
			i	:= i + 1;
		END_IF
	ELSE
		i	:= i + 1;
	END_IF
END_WHILE
END_METHOD

METHOD M_UpdateStatus
VAR_INPUT
END_VAR
// TODO
//
// Copy values from stat.lrReadings to correspondig stat variables
//
// This is an example for model 340.
// This method has to match the list of commands in T_LAKESHORE_CFG::cmdList_Read
stat.lrKRDG_A	:= stat.lrArrReadings[0].lrValue;
stat.lrCRDG_A	:= stat.lrArrReadings[1].lrValue;
stat.lrSETP		:= stat.lrArrReadings[2].lrValue;
stat.nPID_P		:= LREAL_TO_UINT(stat.lrArrReadings[3].lrValue);
stat.nPID_I		:= LREAL_TO_UINT(stat.lrArrReadings[4].lrValue);
stat.nPID_D		:= LREAL_TO_UINT(stat.lrArrReadings[5].lrValue);
stat.bRAMP_On	:= LREAL_TO_BOOL(stat.lrArrReadings[6].lrValue);
stat.lrRAMP_Rate:= stat.lrArrReadings[7].lrValue;
stat.lrKRDG_B	:= stat.lrArrReadings[8].lrValue;
stat.lrCRDG_B	:= stat.lrArrReadings[9].lrValue;
stat.nRANGE		:= LREAL_TO_UINT(stat.lrArrReadings[10].lrValue);
stat.lrHTR		:= stat.lrArrReadings[11].lrValue;
END_METHOD

METHOD ProcessEvents
VAR_INPUT
END_VAR

(* 
	Before processing the event, execute the Do-Activity tasks. 
	Note that, in case of orthogonal regions, more than one Do-Activity 
	could run in the same PLC cycle.
	Note: Most of these activities have timeouts since they take time.
*)

IF	statRef.nSubstate = E_RS_BASE_SUBSTATE.OP_MONITORING 		OR 
	statRef.nSubstate = E_RS_BASE_SUBSTATE.NOTOP_READY			OR
	(statRef.nSubstate = E_RS_BASE_SUBSTATE.NOTOP_ERROR 	AND 
	 nLastGoodSubstate = E_RS_BASE_SUBSTATE.NOTOP_READY) 		OR 
	(statRef.nSubstate = E_RS_BASE_SUBSTATE.OP_ERROR 		AND 
	 nLastGoodSubstate = E_RS_BASE_SUBSTATE.OP_MONITORING)			THEN
	ActivityMonitoring(TRUE);
ELSIF statRef.nSubstate = E_RS_BASE_SUBSTATE.OP_MONITORING_USER THEN
	ActivityMonitoringUser(TRUE);
ELSIF statRef.nSubstate = E_RS_BASE_SUBSTATE.NOTOP_INITIALIZING THEN
	ActivityInitializing(TRUE);
END_IF

// Set last known good substate. Used for recovery from comm problems.
M_SetLastGoodSubstate();

(* 
	Evaluate state machine transitions.
*)

CASE statRef.nState OF

//***********************************
// NOTOP
//***********************************
E_RS_BASE_STATE.NOTOP:

	(* Transitions from NOTOP substates *)
	CASE statRef.nSubstate OF
	
	E_RS_BASE_SUBSTATE.NOTOP_NOTREADY:		
		IF 	nEvent = E_SM_EVENT.INIT OR cfgRef.bAutoMonitor  THEN
			nEvent := E_SM_EVENT.INIT;
			ActionInitExecute();
			SetState(E_RS_BASE_STATE.NOTOP, E_RS_BASE_SUBSTATE.NOTOP_INITIALIZING);
			SetStatus(E_SM_ERROR.OK, 'OK');
			RETURN;
		END_IF
		
	E_RS_BASE_SUBSTATE.NOTOP_INITIALIZING:			
		IF nEvent = E_SM_EVENT.INITDONE THEN
			nReadType := E_RS_BASE_READ_TYPE.PERIODIC;
			ActivityMonitoring(FALSE);	// Reset Monitoring method
			IF cfgRef.bAutoMonitor THEN
				nEvent := E_SM_EVENT.ENABLE;
				statRef.bAutoStarted	:= TRUE;
				SetState(E_RS_BASE_STATE.OP, E_RS_BASE_SUBSTATE.OP_MONITORING);
			ELSE
				SetState(E_RS_BASE_STATE.NOTOP, E_RS_BASE_SUBSTATE.NOTOP_READY);
			END_IF
			RETURN;
		ELSIF nEvent = E_SM_EVENT.ERRINIT THEN
			// INIT failed. Keep re-trying.
			SetState(E_RS_BASE_STATE.NOTOP, E_RS_BASE_SUBSTATE.NOTOP_NOTREADY);
			RETURN;
		END_IF
		
	E_RS_BASE_SUBSTATE.NOTOP_READY:			
		IF nEvent = E_SM_EVENT.ENABLE THEN
			IF cfgRef.bAutoMonitor THEN
				// Monitoring is already in progress.
				// It has to complete the read cycle in a clean way.
				nNextState		:= E_RS_BASE_STATE.OP;					// Next state after STOP	
				nNextSubstate	:= E_RS_BASE_SUBSTATE.OP_MONITORING;	// Next substate after STOP	
				nNextDescription:= 'BUSY';
				nReadType		:= E_RS_BASE_READ_TYPE.PERIODIC;
				RETURN;
			ELSE
				SetState(E_RS_BASE_STATE.OP, E_RS_BASE_SUBSTATE.OP_MONITORING);
				// This call MUST be after SetState()
				ActivityMonitoring(FALSE);	// Reset Monitoring method
			END_IF
		END_IF

	E_RS_BASE_SUBSTATE.NOTOP_ERROR:			
		IF nEvent = E_SM_EVENT.HWOK THEN
			SetState(E_RS_BASE_STATE.NOTOP, E_RS_BASE_SUBSTATE.NOTOP_NOTREADY);
			RETURN;
		ELSIF nEvent = E_SM_EVENT.COMMOK THEN
			SetState(E_RS_BASE_STATE.NOTOP, nLastGoodSubstate);
			RETURN;			
		END_IF
		
	END_CASE

	(* Transitions from NOTOP state *)
	IF	nEvent = E_SM_EVENT.ERRHW OR
		nEvent = E_SM_EVENT.ERRCOMM	THEN
		ActionUnexpExecute();
		SetState(E_RS_BASE_STATE.NOTOP, E_RS_BASE_SUBSTATE.NOTOP_ERROR);
		RETURN;
	END_IF
	
//***********************************
// OPERATIONAL
//***********************************
E_RS_BASE_STATE.OP:

	(* Transitions from OP subastates *)
	CASE statRef.nSubstate OF
	E_RS_BASE_SUBSTATE.OP_ERROR:			
		IF 	cfgRef.bAutoMonitor  THEN
			nEvent := E_SM_EVENT.INIT;
			ActionInitExecute();
			SetState(E_RS_BASE_STATE.NOTOP, E_RS_BASE_SUBSTATE.NOTOP_INITIALIZING);
			SetStatus(E_SM_ERROR.OK, 'Recovering from error...');
			RETURN;
		END_IF
		IF nEvent = E_SM_EVENT.HWOK THEN
			SetStatus(E_SM_ERROR.OK, 'OK');
			SetState(E_RS_BASE_STATE.OP, E_RS_BASE_SUBSTATE.OP_IDLE);
			RETURN;			
		ELSIF nEvent = E_SM_EVENT.DISABLE THEN
			ActionDisableExecute();
			SetState(E_RS_BASE_STATE.NOTOP, E_RS_BASE_SUBSTATE.NOTOP_ERROR);
			RETURN;			
		ELSIF nEvent = E_SM_EVENT.COMMOK THEN
			SetState(E_RS_BASE_STATE.OP, nLastGoodSubstate);
			RETURN;			
		END_IF

	E_RS_BASE_SUBSTATE.OP_MONITORING:
		IF nEvent = E_SM_EVENT.DISABLE THEN
			ActionDisableExecute();
			RETURN;			
		ELSIF nEvent = E_SM_EVENT.STOPMON THEN
			ActionStopExecute();
			RETURN;			
		ELSIF nEvent = E_SM_EVENT.READDONE THEN
			SetState(E_RS_BASE_STATE.OP, E_RS_BASE_SUBSTATE.OP_IDLE);
			RETURN;			
		ELSIF nEvent = E_SM_EVENT.ERRCOMM THEN
			SetState(E_RS_BASE_STATE.OP, E_RS_BASE_SUBSTATE.OP_ERROR);
			RETURN;			
		END_IF
		
	E_RS_BASE_SUBSTATE.OP_MONITORING_USER:			
		IF nEvent = E_SM_EVENT.DISABLE THEN
			ActionDisableExecute();
			RETURN;			
		ELSIF nEvent = E_SM_EVENT.STOPMON THEN
			ActionStopExecute();
			RETURN;			
		ELSIF nEvent = E_SM_EVENT.READDONE THEN
			SetState(E_RS_BASE_STATE.OP, E_RS_BASE_SUBSTATE.OP_IDLE);
			RETURN;			
		END_IF
		
	E_RS_BASE_SUBSTATE.OP_IDLE:			
		IF nEvent = E_SM_EVENT.DISABLE THEN
			ActionDisableExecute();
			RETURN;			
		ELSIF nEvent = E_SM_EVENT.READ THEN
			nReadType	:= E_RS_BASE_READ_TYPE.SINGLE;
			ActivityMonitoring(FALSE);	// Reset Monitoring method
			SetState(E_RS_BASE_STATE.OP, E_RS_BASE_SUBSTATE.OP_MONITORING);
			RETURN;			
		ELSIF nEvent = E_SM_EVENT.READ_USER THEN
			nReadType	:= E_RS_BASE_READ_TYPE.SINGLE_USER;
			ActivityMonitoringUser(FALSE);	// Reset Monitoring method
			SetState(E_RS_BASE_STATE.OP, E_RS_BASE_SUBSTATE.OP_MONITORING_USER);
			RETURN;			
		ELSIF nEvent = E_SM_EVENT.MONITOR OR nEvent = E_SM_EVENT.ENABLE THEN
			nReadType	:= E_RS_BASE_READ_TYPE.PERIODIC;
			ActivityMonitoring(FALSE);	// Reset Monitoring method
			SetState(E_RS_BASE_STATE.OP, E_RS_BASE_SUBSTATE.OP_MONITORING);
			RETURN;			
		ELSIF nEvent = E_SM_EVENT.MONITOR_USER THEN
			nReadType	:= E_RS_BASE_READ_TYPE.PERIODIC_USER;
			ActivityMonitoringUser(FALSE);	// Reset Monitoring method
			SetState(E_RS_BASE_STATE.OP, E_RS_BASE_SUBSTATE.OP_MONITORING_USER);
			RETURN;			
		END_IF
		
	END_CASE
	
	// Transitions from OP state.
	// Valid for any OP substate.
	IF nEvent = E_SM_EVENT.ERRHW THEN
		ActionUnexpExecute();
		SetState(E_RS_BASE_STATE.OP, E_RS_BASE_SUBSTATE.OP_ERROR);
		RETURN;
	ELSIF nEvent = E_SM_EVENT.ERRCOMM THEN
		SetState(E_RS_BASE_STATE.OP, E_RS_BASE_SUBSTATE.OP_ERROR);
		RETURN;
	END_IF
	
END_CASE

(* 
	"Global" internal transitions valid in any state should go here.
	They do not change the active state configuration. 
	They are evaluated after all the others transitions have been 
	considered.
*) 
IF nEvent = E_SM_EVENT.RESET THEN
	ActionResetExecute();
	SetState(E_RS_BASE_STATE.NOTOP, E_RS_BASE_SUBSTATE.NOTOP_NOTREADY);
	RETURN;
END_IF
END_METHOD

END_FUNCTION_BLOCK

// POUs/FB_RS_BASE
FUNCTION_BLOCK FB_RS_BASE
VAR_INPUT
	{attribute 'OPC.UA.DA' := '0'}
	in_bSimulation:	BOOL := FALSE;
	{attribute 'OPC.UA.DA' := '0'}
	in_sName:		STRING := 'RS Dev';	// Instance name
END_VAR
VAR_OUTPUT
END_VAR
VAR RETAIN
END_VAR
VAR
	{attribute 'OPC.UA.DA' := '0'}
	cfgRef:			REFERENCE TO T_RS_BASE_CFG;	
	{attribute 'OPC.UA.DA' := '0'}
	ctrlRef:		REFERENCE TO T_RS_BASE_CTRL;	
	{attribute 'OPC.UA.DA' := '0'}
	statRef:		REFERENCE TO T_RS_BASE_STAT;	// Common State Machine Status - ReadOnly 

	{attribute 'OPC.UA.DA' := '0'}
	nEvent:		      	DINT := E_SM_EVENT.NONE;
	{attribute 'OPC.UA.DA' := '0'}
	nInternalEvent:		DINT := E_SM_EVENT.NONE;
	
	{attribute 'OPC.UA.DA' := '0'}
	nNextState:			E_RS_BASE_STATE		:= E_RS_BASE_STATE.NONE;		// Next state after STOP	
	{attribute 'OPC.UA.DA' := '0'}
	nNextSubstate:		E_RS_BASE_SUBSTATE	:= E_RS_BASE_SUBSTATE.NONE;	// Next substate after STOP	
	{attribute 'OPC.UA.DA' := '0'}
	nNextDescription:	STRING			:= '';					// Next substate description	
	
	{attribute 'OPC.UA.DA' := '0'}
	nReadType:		E_RS_BASE_READ_TYPE;
	
	{attribute 'OPC.UA.DA' := '0'}
	bCommProblem:	BOOL := FALSE;	// Flag if there is a communication problem
	{attribute 'OPC.UA.DA' := '0'}
	nLastGoodSubstate:	INT	:= E_RS_BASE_SUBSTATE.NONE;	// Used for recovery

END_VAR

// Don't do anything in the first 100 cycles in order for the system to stabilise.
statRef.nCycleCounter	:= statRef.nCycleCounter + 1;
IF statRef.bActive AND statRef.nCycleCounter < 100 THEN
	RETURN;
ELSE
	statRef.bActive	:= TRUE;
END_IF


// Set simulation flag in the status structure
statRef.bSimulation	:= in_bSimulation;


(* === Check for commands and internal events to be processed === *)
CheckForEvents();

(* === Process events according to the State Machine === *)
ProcessEvents();

METHOD ActionDisableExecute
VAR_INPUT
END_VAR
SetAction('ActionDisableExecute');

IF statRef.nSubstate =E_RS_BASE_SUBSTATE.OP_IDLE 	THEN
	SetState(E_RS_BASE_STATE.NOTOP, E_RS_BASE_SUBSTATE.NOTOP_READY);
ELSE		
	nNextState		:= E_RS_BASE_STATE.NOTOP;			// Next state after STOP	
	nNextSubstate	:= E_RS_BASE_SUBSTATE.NOTOP_READY;	// Next substate after STOP	
	nNextDescription:= 'BUSY';
END_IF
END_METHOD

METHOD ActionEnableExecute
VAR_INPUT
END_VAR
END_METHOD

METHOD ActionErrExecute
VAR_INPUT
END_VAR
SetAction('ActionErrExecute');

IF nEvent = E_SM_EVENT.ERRHW THEN
	SetStatus(E_SM_ERROR.HW_NOT_OP, 'ERROR: HW not in OP state');	
ELSIF nEvent = E_SM_EVENT.ERRINIT THEN
	SetStatus(E_SM_ERROR.INIT_FAILURE, 'ERROR: INIT failed');	
END_IF
END_METHOD

METHOD ActionInitExecute
VAR_INPUT
END_VAR
SetAction('ActionInitExecute');

ActivityInitializing(FALSE);
END_METHOD

METHOD ActionResetExecute
VAR_INPUT
END_VAR
SetAction('ActionResetExecute');

// TODO
//nEvent := E_SM_EVENT.NONE;

// Clear error
SetStatus(E_SM_ERROR.OK, 'OK');
END_METHOD

METHOD ActionStopExecute
VAR_INPUT
END_VAR
SetAction('ActionStopExecute');

IF statRef.nSubstate = E_RS_BASE_SUBSTATE.NOTOP_READY 	THEN
	RETURN;
ELSE		
	nNextState		:= E_RS_BASE_STATE.OP;			// Next state after STOP	
	nNextSubstate	:= E_RS_BASE_SUBSTATE.OP_IDLE;	// Next substate after STOP	
	nNextDescription:= 'IDLE';
END_IF
END_METHOD

METHOD ActionUnexpExecute
VAR_INPUT
END_VAR
SetAction('ActionUnexpExecute');

(*
	We don't want to overwrite initial error.
	Update error only if it is currently equal to OK. 
*)
IF statRef.nErrorCode = E_SM_ERROR.OK THEN
	IF nEvent = E_SM_EVENT.ERRHW THEN
		statRef.nErrorCode		:= E_SM_ERROR.HW_NOT_OP;
		statRef.sErrorText		:= 'ERROR: HW not in OP state.';	
	ELSIF nEvent = E_SM_EVENT.ERRINIT THEN
		statRef.nErrorCode		:= E_SM_ERROR.INIT_FAILURE;
		statRef.sErrorText		:= 'ERROR: INIT failed.';	
	END_IF
END_IF
END_METHOD

METHOD ActivityInitializing
VAR_INPUT
	bExecute:	BOOL;
END_VAR
SetAction('ActivityInitializing');

IF	NOT M_GetCouplerState()  THEN
	nInternalEvent 		:= E_SM_EVENT.ERRHW;

	SetStatus(E_SM_ERROR.HW_NOT_OP, 'HW not in OP state');	
	RETURN;
END_IF
END_METHOD

METHOD ActivityMonitoring
VAR_INPUT
	bExecute:	BOOL;
END_VAR
SetAction('ActivityMonitoring');
END_METHOD

METHOD ActivityMonitoringUser
VAR_INPUT
	bExecute:	BOOL;
END_VAR
SetAction('ActivityMonitoringUser');
END_METHOD

METHOD CheckForEvents
VAR_INPUT
END_VAR
VAR
END_VAR

(* 
	Start assuming the HW is OK in case there was no communication problem. 
	This is needed to recover from the situation where 
	the HW was failing and now it is working.
*)

//IF NOT bCommProblem	THEN
//	nInternalEvent := E_SM_EVENT.HWOK;
//END_IF




(* 
	Check for events in the following order: 
   	1) HW failure: without HW avilability there is no point to do anything
	2) Internal events: to allow completing the initiated commands before 
                        starting processing new commands. 
   	3) Commands: to react to external commands. Commands should be executed 
                 before processing HW signals to allow to start a recovery action.
   	4) HW signals: if any.
*)

IF NOT M_GetCouplerState() THEN	
	(* Check if the HW is NOT OK *)
	(*
	If the hardware status is NOT OK, we cannot trust the readings.
	Variable i_nCouplerState has to be mapped to a State of a terminal, e.g. EK1100.
	The value should be 8.
 	*)
	SetEvent(E_SM_EVENT.ERRHW);
	SetStatus(E_SM_ERROR.HW_NOT_OP, 'ERROR: HW not in OPERATIONAL state');

ELSIF ctrlRef.bExecute  THEN
	(* Handle commands *)
	ctrlRef.bExecute		:= FALSE;			(* Clear the Execute bit *)
	SetLastCommand(ctrlRef.nCommand);			(* Save the last command *)
	SetEvent(ctrlRef.nCommand);
	ctrlRef.nCommand 		:= E_RS_COMMAND.NONE;	(* Clear the Command *)
ELSIF nInternalEvent <> E_SM_EVENT.NONE THEN
	(* Handle internal events *)
	SetEvent(nInternalEvent);
	nInternalEvent := E_SM_EVENT.NONE;
ELSE
	(* Handle HW problems and unexpected bahaviour *)
	
END_IF
END_METHOD

METHOD M_Configure
VAR_INPUT
END_VAR
END_METHOD

METHOD M_GetCouplerState : BOOL
VAR_INPUT
END_VAR
M_GetCouplerState	:= true;
END_METHOD

METHOD M_GetRpcErrorText : STRING
VAR_INPUT
	ErrorCode:	INT;
END_VAR
VAR
	str:	STRING;
END_VAR
CASE ErrorCode OF
	E_RS_RPC_ERROR.OK:					str	:= 'OK';
	E_RS_RPC_ERROR.NOT_OP:				str	:= 'Cannot control device. Not in OP state.';
	E_RS_RPC_ERROR.NOT_NOTOP_READY:		str	:= 'Call failed. Not in NOTOP_READY.';
	E_RS_RPC_ERROR.NOT_NOTOP_NOTREADY:	str	:= 'Call failed. Not in NOTOP_NOTREADY/ERROR.';
	E_RS_RPC_ERROR.LOCAL:				str	:= 'RPC calls not allowed in Local mode.';
ELSE
	str	:= 'Unregistered RPC error.';
END_CASE

M_GetRpcErrorText	:= str;
END_METHOD

METHOD M_ReadSensors
VAR_INPUT
END_VAR
END_METHOD

METHOD M_SetLastGoodSubstate
VAR_INPUT
END_VAR
IF	statRef.nSubstate <> E_RS_BASE_SUBSTATE.NOTOP_ERROR	AND 
	statRef.nSubstate <> E_RS_BASE_SUBSTATE.OP_ERROR			THEN
	nLastGoodSubstate := statRef.nSubstate;			
END_IF
END_METHOD

METHOD M_SetRpcStatus : INT
VAR_INPUT
	nErrorCode:	INT;
END_VAR
statRef.nRpcErrorCode	:= nErrorCode;
statRef.sRpcErrorText	:= M_GetRpcErrorText(nErrorCode);

M_SetRpcStatus		:= nErrorCode;
END_METHOD

METHOD ProcessEvents
VAR_INPUT
END_VAR

(* 
	Before processing the event, execute the Do-Activity tasks. 
	Note that, in case of orthogonal regions, more than one Do-Activity 
	could run in the same PLC cycle.
	Note: Most of these activities have timeouts since they take time.
*)

IF	statRef.nSubstate = E_RS_BASE_SUBSTATE.OP_MONITORING 		OR 
	statRef.nSubstate = E_RS_BASE_SUBSTATE.NOTOP_READY			OR
	(statRef.nSubstate = E_RS_BASE_SUBSTATE.NOTOP_ERROR 	AND 
	 nLastGoodSubstate = E_RS_BASE_SUBSTATE.NOTOP_READY) 		OR 
	(statRef.nSubstate = E_RS_BASE_SUBSTATE.OP_ERROR 		AND 
	 nLastGoodSubstate = E_RS_BASE_SUBSTATE.OP_MONITORING)			THEN
	ActivityMonitoring(TRUE);
ELSIF statRef.nSubstate = E_RS_BASE_SUBSTATE.OP_MONITORING_USER THEN
	ActivityMonitoringUser(TRUE);
ELSIF statRef.nSubstate = E_RS_BASE_SUBSTATE.NOTOP_INITIALIZING THEN
	ActivityInitializing(TRUE);
END_IF

// Set last known good substate. Used for recovery from comm problems.
M_SetLastGoodSubstate();

(* 
	Evaluate state machine transitions.
*)

CASE statRef.nState OF

//***********************************
// NOTOP
//***********************************
E_RS_BASE_STATE.NOTOP:

	(* Transitions from NOTOP substates *)
	CASE statRef.nSubstate OF
	
	E_RS_BASE_SUBSTATE.NOTOP_NOTREADY:		
		IF 	nEvent = E_SM_EVENT.INIT OR 
			(cfgRef.bAutoMonitor AND NOT statRef.bAutoStarted)  THEN
			nEvent := E_SM_EVENT.INIT;
			ActionInitExecute();
			SetState(E_RS_BASE_STATE.NOTOP, E_RS_BASE_SUBSTATE.NOTOP_INITIALIZING);
			SetStatus(E_SM_ERROR.OK, 'OK');
			RETURN;
		END_IF
		
	E_RS_BASE_SUBSTATE.NOTOP_INITIALIZING:			
		IF nEvent = E_SM_EVENT.INITDONE THEN
			nReadType := E_RS_BASE_READ_TYPE.PERIODIC;
			ActivityMonitoring(FALSE);	// Reset Monitoring method
			IF cfgRef.bAutoMonitor THEN
				nEvent := E_SM_EVENT.ENABLE;
				statRef.bAutoStarted	:= TRUE;
				SetState(E_RS_BASE_STATE.OP, E_RS_BASE_SUBSTATE.OP_MONITORING);
			ELSE
				SetState(E_RS_BASE_STATE.NOTOP, E_RS_BASE_SUBSTATE.NOTOP_READY);
			END_IF
			RETURN;
		ELSIF nEvent = E_SM_EVENT.ERRINIT THEN
			statRef.bAutoStarted	:= TRUE;
			SetState(E_RS_BASE_STATE.NOTOP, E_RS_BASE_SUBSTATE.NOTOP_NOTREADY);
			RETURN;
		END_IF
		
	E_RS_BASE_SUBSTATE.NOTOP_READY:			
		IF nEvent = E_SM_EVENT.ENABLE THEN
			IF cfgRef.bAutoMonitor THEN
				// Monitoring is already in progress.
				// It has to complete the read cycle in a clean way.
				nNextState		:= E_RS_BASE_STATE.OP;					// Next state after STOP	
				nNextSubstate	:= E_RS_BASE_SUBSTATE.OP_MONITORING;	// Next substate after STOP	
				nNextDescription:= 'BUSY';
				nReadType		:= E_RS_BASE_READ_TYPE.PERIODIC;
				RETURN;
			ELSE
				SetState(E_RS_BASE_STATE.OP, E_RS_BASE_SUBSTATE.OP_MONITORING);
				// This call MUST be after SetState()
				ActivityMonitoring(FALSE);	// Reset Monitoring method
			END_IF
		END_IF

	E_RS_BASE_SUBSTATE.NOTOP_ERROR:			
		IF nEvent = E_SM_EVENT.HWOK THEN
			SetState(E_RS_BASE_STATE.NOTOP, E_RS_BASE_SUBSTATE.NOTOP_NOTREADY);
			RETURN;
		ELSIF nEvent = E_SM_EVENT.COMMOK THEN
			SetState(E_RS_BASE_STATE.NOTOP, nLastGoodSubstate);
			RETURN;			
		END_IF
		
	END_CASE

	(* Transitions from NOTOP state *)
	IF	nEvent = E_SM_EVENT.ERRHW OR
		nEvent = E_SM_EVENT.ERRCOMM	THEN
		ActionUnexpExecute();
		SetState(E_RS_BASE_STATE.NOTOP, E_RS_BASE_SUBSTATE.NOTOP_ERROR);
		RETURN;
	END_IF
	
//***********************************
// OPERATIONAL
//***********************************
E_RS_BASE_STATE.OP:

	(* Transitions from OP subastates *)
	CASE statRef.nSubstate OF
	E_RS_BASE_SUBSTATE.OP_ERROR:			
		IF 	cfgRef.bAutoMonitor  THEN
			nEvent := E_SM_EVENT.INIT;
			ActionInitExecute();
			SetState(E_RS_BASE_STATE.NOTOP, E_RS_BASE_SUBSTATE.NOTOP_INITIALIZING);
			SetStatus(E_SM_ERROR.OK, 'Recovering from error...');
			RETURN;
		END_IF
		IF nEvent = E_SM_EVENT.HWOK THEN
			SetStatus(E_SM_ERROR.OK, 'OK');
			SetState(E_RS_BASE_STATE.OP, E_RS_BASE_SUBSTATE.OP_IDLE);
			RETURN;			
		ELSIF nEvent = E_SM_EVENT.DISABLE THEN
			ActionDisableExecute();
			SetState(E_RS_BASE_STATE.NOTOP, E_RS_BASE_SUBSTATE.NOTOP_ERROR);
			RETURN;			
		ELSIF nEvent = E_SM_EVENT.COMMOK THEN
			SetState(E_RS_BASE_STATE.OP, nLastGoodSubstate);
			RETURN;			
		END_IF

	E_RS_BASE_SUBSTATE.OP_MONITORING:
		IF nEvent = E_SM_EVENT.DISABLE THEN
			ActionDisableExecute();
			RETURN;			
		ELSIF nEvent = E_SM_EVENT.STOPMON THEN
			ActionStopExecute();
			RETURN;			
		ELSIF nEvent = E_SM_EVENT.READDONE THEN
			SetState(E_RS_BASE_STATE.OP, E_RS_BASE_SUBSTATE.OP_IDLE);
			RETURN;			
		ELSIF nEvent = E_SM_EVENT.ERRCOMM THEN
			SetState(E_RS_BASE_STATE.OP, E_RS_BASE_SUBSTATE.OP_ERROR);
			RETURN;			
		END_IF
		
	E_RS_BASE_SUBSTATE.OP_MONITORING_USER:			
		IF nEvent = E_SM_EVENT.DISABLE THEN
			ActionDisableExecute();
			RETURN;			
		ELSIF nEvent = E_SM_EVENT.STOPMON THEN
			ActionStopExecute();
			RETURN;			
		ELSIF nEvent = E_SM_EVENT.READDONE THEN
			SetState(E_RS_BASE_STATE.OP, E_RS_BASE_SUBSTATE.OP_IDLE);
			RETURN;			
		END_IF
		
	E_RS_BASE_SUBSTATE.OP_IDLE:			
		IF nEvent = E_SM_EVENT.DISABLE THEN
			ActionDisableExecute();
			RETURN;			
		ELSIF nEvent = E_SM_EVENT.READ THEN
			nReadType	:= E_RS_BASE_READ_TYPE.SINGLE;
			ActivityMonitoring(FALSE);	// Reset Monitoring method
			SetState(E_RS_BASE_STATE.OP, E_RS_BASE_SUBSTATE.OP_MONITORING);
			RETURN;			
		ELSIF nEvent = E_SM_EVENT.READ_USER THEN
			nReadType	:= E_RS_BASE_READ_TYPE.SINGLE_USER;
			ActivityMonitoringUser(FALSE);	// Reset Monitoring method
			SetState(E_RS_BASE_STATE.OP, E_RS_BASE_SUBSTATE.OP_MONITORING_USER);
			RETURN;			
		ELSIF nEvent = E_SM_EVENT.MONITOR OR nEvent = E_SM_EVENT.ENABLE THEN
			nReadType	:= E_RS_BASE_READ_TYPE.PERIODIC;
			ActivityMonitoring(FALSE);	// Reset Monitoring method
			SetState(E_RS_BASE_STATE.OP, E_RS_BASE_SUBSTATE.OP_MONITORING);
			RETURN;			
		ELSIF nEvent = E_SM_EVENT.MONITOR_USER THEN
			nReadType	:= E_RS_BASE_READ_TYPE.PERIODIC_USER;
			ActivityMonitoringUser(FALSE);	// Reset Monitoring method
			SetState(E_RS_BASE_STATE.OP, E_RS_BASE_SUBSTATE.OP_MONITORING_USER);
			RETURN;			
		END_IF
		
	END_CASE
	
	// Transitions from OP state.
	// Valid for any OP substate.
	IF nEvent = E_SM_EVENT.ERRHW THEN
		ActionUnexpExecute();
		SetState(E_RS_BASE_STATE.OP, E_RS_BASE_SUBSTATE.OP_ERROR);
		RETURN;
	ELSIF nEvent = E_SM_EVENT.ERRCOMM THEN
		SetState(E_RS_BASE_STATE.OP, E_RS_BASE_SUBSTATE.OP_ERROR);
		RETURN;
	END_IF
	
END_CASE

(* 
	"Global" internal transitions valid in any state should go here.
	They do not change the active state configuration. 
	They are evaluated after all the others transitions have been 
	considered.
*) 
IF nEvent = E_SM_EVENT.RESET THEN
	ActionResetExecute();
	SetState(E_RS_BASE_STATE.NOTOP, E_RS_BASE_SUBSTATE.NOTOP_NOTREADY);
	RETURN;
END_IF
END_METHOD

{attribute 'TcRpcEnable':='1'}
METHOD RPC_Disable : INT
VAR_INPUT
END_VAR
VAR
END_VAR
// RPC calls are not allowed in Local mode.
IF statRef.bLocal THEN
	RPC_Disable	:= M_SetRpcStatus(E_RS_RPC_ERROR.LOCAL);
	RETURN;
END_IF

// Disable command is accepted only if device is in OP state.
IF statRef.nState <> E_RS_BASE_STATE.OP THEN
	RPC_Disable	:= M_SetRpcStatus(E_RS_RPC_ERROR.NOT_OP);
	RETURN;
ELSE
	ctrlRef.nCommand := E_RS_COMMAND.DISABLE;
	ctrlRef.bExecute := TRUE;
	
	// Call was successful
	RPC_Disable	:= M_SetRpcStatus(E_RS_RPC_ERROR.OK);
END_IF
END_METHOD

{attribute 'TcRpcEnable':='1'}
METHOD RPC_Enable : INT
VAR_INPUT
END_VAR
VAR
END_VAR
// RPC calls are not allowed in Local mode.
IF statRef.bLocal THEN
	RPC_Enable	:= M_SetRpcStatus(E_RS_RPC_ERROR.LOCAL);
	RETURN;
END_IF

// Enable command is accepted only if device is in NOTOP_READY.
// Enable command is ignored (in ProcessEvents) if operational.
IF	statRef.nSubstate <> E_RS_BASE_SUBSTATE.NOTOP_READY			AND
	statRef.nSubstate <> E_RS_BASE_SUBSTATE.OP_MONITORING		AND
	statRef.nSubstate <> E_RS_BASE_SUBSTATE.OP_IDLE				AND
	statRef.nSubstate <> E_RS_BASE_SUBSTATE.OP_MONITORING_USER		THEN
	RPC_Enable	:= M_SetRpcStatus(E_RS_RPC_ERROR.NOT_NOTOP_READY);
	RETURN;
ELSE
	ctrlRef.nCommand := E_RS_COMMAND.ENABLE;
	ctrlRef.bExecute := TRUE;
	
	// Call was successful
	RPC_Enable	:= M_SetRpcStatus(E_RS_RPC_ERROR.OK);
END_IF
END_METHOD

{attribute 'TcRpcEnable':='1'}
METHOD RPC_Init : INT
VAR_INPUT
END_VAR
VAR
END_VAR
// RPC calls are not allowed in Local mode.
IF statRef.bLocal THEN
	RPC_Init	:= M_SetRpcStatus(E_RS_RPC_ERROR.LOCAL);
	RETURN;
END_IF

// Init command is accepted only if device is in NOTOP_NOTREADY or ERROR.
IF 	statRef.nSubstate <> E_RS_BASE_SUBSTATE.NOTOP_NOTREADY  AND  
	statRef.nSubstate <> E_RS_BASE_SUBSTATE.NOTOP_ERROR 		THEN
	RPC_Init	:= M_SetRpcStatus(E_RS_RPC_ERROR.NOT_NOTOP_NOTREADY);
	RETURN;
ELSE
	ctrlRef.nCommand := E_RS_COMMAND.INIT;
	ctrlRef.bExecute := TRUE;
	
	// Call was successful
	RPC_Init	:= M_SetRpcStatus(E_RS_RPC_ERROR.OK);
END_IF
END_METHOD

{attribute 'TcRpcEnable':='1'}
METHOD RPC_Reset : INT
VAR_INPUT
END_VAR
VAR
END_VAR
// RPC calls are not allowed in Local mode.
IF statRef.bLocal THEN
	RPC_Reset	:= M_SetRpcStatus(E_RS_RPC_ERROR.LOCAL);
	RETURN;
END_IF

ctrlRef.nCommand := E_RS_COMMAND.RESET;
ctrlRef.bExecute := TRUE;

// Call was successful
RPC_Reset	:= M_SetRpcStatus(E_RS_RPC_ERROR.OK);
END_METHOD

{attribute 'TcRpcEnable':='1'}
METHOD RPC_Stop : INT
VAR_INPUT
END_VAR
VAR
END_VAR
// RPC calls are not allowed in Local mode.
IF statRef.bLocal THEN
	RPC_Stop	:= M_SetRpcStatus(E_RS_RPC_ERROR.LOCAL);
	RETURN;
END_IF

ctrlRef.nCommand := E_RS_COMMAND.STOP;
ctrlRef.bExecute := TRUE;

// Call was successful
RPC_Stop	:= M_SetRpcStatus(E_RS_RPC_ERROR.OK);
END_METHOD

METHOD SetAction
VAR_INPUT
	actionName:		STRING;
END_VAR


statRef.sActionDesc := actionName;
END_METHOD

METHOD SetEvent
VAR_INPUT
	nEventId:			DINT;
END_VAR

nEvent := nEventId;

CASE nEventId OF
	E_SM_EVENT.NONE:
		statRef.sEventDesc := '';
		RETURN;
		
	E_SM_EVENT.RESET:
		statRef.sEventDesc := 'CMD RESET';
		RETURN;
	
	E_SM_EVENT.INIT:
		statRef.sEventDesc := 'CMD INIT';
		RETURN;

	E_SM_EVENT.STOP:
		statRef.sEventDesc := 'CMD STOP';
		RETURN;

	E_SM_EVENT.ENABLE:
		statRef.sEventDesc := 'CMD ENABLE';
		RETURN;

	E_SM_EVENT.DISABLE:
		statRef.sEventDesc := 'CMD DISABLE';
		RETURN;

		
	E_SM_EVENT.READ:
		statRef.sEventDesc := 'CMD SINGLE READ';
		RETURN;

	E_SM_EVENT.READ_USER:
		statRef.sEventDesc := 'CMD SINGLE READ USER';
		RETURN;

	E_SM_EVENT.MONITOR:
		statRef.sEventDesc := 'CMD MONITOR';
		RETURN;

	E_SM_EVENT.MONITOR_USER:
		statRef.sEventDesc := 'CMD MONITOR USER';
		RETURN;

	E_SM_EVENT.STOPMON:
		statRef.sEventDesc := 'CMD STOP MONITOR';
		RETURN;

	E_SM_EVENT.CTRL_CMD:
		statRef.sEventDesc := 'CMD CTRL_CMD';
		RETURN;


	(* events corresponding to internal events *)
	(* events mapped to HW signals *)
	E_SM_EVENT.INITDONE:
		statRef.sEventDesc := 'INT INITDONE';
		RETURN;

	E_SM_EVENT.READDONE:
		statRef.sEventDesc := 'INT READDONE';
		RETURN;

	E_SM_EVENT.HWOK:
		statRef.sEventDesc := 'SIG HWOK';
		RETURN;

	E_SM_EVENT.COMMOK:
		statRef.sEventDesc := 'SIG COMMOK';
		RETURN;

	E_SM_EVENT.ERRCOMM:
		statRef.sEventDesc := 'INT ERRCOMM';
		RETURN;

	E_SM_EVENT.ERRHW:
		statRef.sEventDesc := 'INT ERRHW';
		RETURN;

	E_SM_EVENT.ERRINIT:
		statRef.sEventDesc := 'INT ERRINIT';
		RETURN;

	
END_CASE 

(* INTERNAL ERROR *)
statRef.sEventDesc := 'UNKNOWN EVENT';
END_METHOD

METHOD SetLastCommand
VAR_INPUT
	cmd:	E_RS_COMMAND;
END_VAR
statRef.nLastCommand	:= cmd;

CASE cmd OF
	E_RS_COMMAND.RESET:
		statRef.sLastCommand	:= 'RESET';
	E_RS_COMMAND.INIT:
		statRef.sLastCommand	:= 'INIT';
	E_RS_COMMAND.STOP:
		statRef.sLastCommand	:= 'STOP';
	E_RS_COMMAND.ENABLE:
		statRef.sLastCommand	:= 'ENABLE';
	E_RS_COMMAND.DISABLE:
		statRef.sLastCommand	:= 'DISABLE';
	E_RS_COMMAND.CTRL_CMD:
		statRef.sLastCommand	:= 'CTRL CMD';
ELSE
		statRef.sLastCommand	:= 'NONE';
END_CASE;
END_METHOD

METHOD SetState
VAR_INPUT
	nState:			INT;
	nSubstate:		INT;
END_VAR
(* 
	Update State Machine active state configuration.

	ToDo: support initial pseudo state/substate.
*)

IF nState <> E_RS_BASE_STATE.NONE THEN
	statRef.nState	:= nState;
END_IF
IF nSubstate <> E_RS_BASE_SUBSTATE.NONE THEN
	statRef.nSubstate	:= nSubstate;
END_IF

(* Update active state configuration description *)

IF nState = E_RS_BASE_STATE.NOTOP THEN
	statRef.sState	:= 'NOT OP';
ELSIF nState = E_RS_BASE_STATE.OP THEN
	statRef.sState	:= 'OPERATIONAL';
END_IF

IF nSubstate = E_RS_BASE_SUBSTATE.NOTOP_NOTREADY THEN
	statRef.sSubstate	:= 'NOT READY';
ELSIF nSubstate = E_RS_BASE_SUBSTATE.NOTOP_INITIALIZING THEN
	statRef.sSubstate	:= 'INITIALIAZING';
ELSIF nSubstate = E_RS_BASE_SUBSTATE.NOTOP_READY THEN
	statRef.sSubstate	:= 'READY';
ELSIF nSubstate = E_RS_BASE_SUBSTATE.NOTOP_ERROR THEN
	statRef.sSubstate	:= 'ERROR';
ELSIF nSubstate = E_RS_BASE_SUBSTATE.OP_MONITORING THEN
	statRef.sSubstate	:= 'MONITORING';
ELSIF nSubstate = E_RS_BASE_SUBSTATE.OP_MONITORING_USER THEN
	statRef.sSubstate	:= 'MONITORING USER';
ELSIF nSubstate = E_RS_BASE_SUBSTATE.OP_IDLE THEN
	statRef.sSubstate	:= 'IDLE';
ELSIF nSubstate = E_RS_BASE_SUBSTATE.OP_ERROR THEN
	statRef.sSubstate	:= 'ERROR';
ELSE
	statRef.sSubstate	:= '';
END_IF
END_METHOD

METHOD SetStatus
VAR_INPUT
	nErrorCode:	INT;
	sErrorText:	STRING;
END_VAR
statRef.nErrorCode 	:= nErrorCode;
statRef.sErrorText 	:= sErrorText;

IF nErrorCode <> E_SM_ERROR.OK THEN
	statRef.sStatus	:= 'ERROR';
	statRef.nStatus	:= E_SM_STATUS.ERROR;
ELSE
	statRef.sStatus	:= 'OK';
	statRef.nStatus	:= E_SM_STATUS.OK;
END_IF
END_METHOD

END_FUNCTION_BLOCK

// POUs/FB_SIM_MODBUS_COMM_BASE
FUNCTION_BLOCK FB_SIM_MODBUS_COMM_BASE
VAR_INPUT
	in_nModel:			DINT;
END_VAR
VAR_OUTPUT
END_VAR
VAR
END_VAR

M_ActivityDo();

METHOD M_ActivityDo
VAR_INPUT
END_VAR
END_METHOD

METHOD M_ByteSwap_INT_TO_BYTES : ARRAY [0..1] OF BYTE
VAR_INPUT
	nValue:	INT;
END_VAR
VAR
	pByte:		POINTER TO BYTE;	// Pointer to nValue
	sResult:	ARRAY [0..1] OF BYTE;
END_VAR
pByte	:= ADR(nValue);

sResult[0]	:= pByte[1];
sResult[1]	:= pByte[0];

M_ByteSwap_INT_TO_BYTES	:= sResult;
END_METHOD

METHOD M_ByteSwap_INT_TO_STRING : STRING
VAR_INPUT
	nValue:	INT;
END_VAR
VAR
	pByte:		POINTER TO BYTE;	// Pointer to nValue
	sResult:	STRING(8) := '';
END_VAR
pByte	:= ADR(nValue);

sResult[0]	:= pByte[1];
sResult[1]	:= pByte[0];

M_ByteSwap_INT_TO_STRING	:= sResult;
END_METHOD

METHOD M_ByteSwap_REAL_TO_BYTES : ARRAY [0..3] OF BYTE
VAR_INPUT
	rValue:		REAL;	// Pointer to real number
END_VAR
VAR
	pByte:		POINTER TO BYTE;	// Pointer to real number
	sResult:	ARRAY [0..3] OF BYTE;
END_VAR
pByte	:= ADR(rValue);

sResult[0]	:= pByte[1];
sResult[1]	:= pByte[0];
sResult[2]	:= pByte[3];
sResult[3]	:= pByte[2];

M_ByteSwap_REAL_TO_BYTES	:= sResult;
END_METHOD

METHOD M_ByteSwap_REAL_TO_STRING : STRING
VAR_INPUT
	rValue:		REAL;	// Pointer to real number
END_VAR
VAR
	pByte:		POINTER TO BYTE;	// Pointer to real number
	sResult:	STRING(8) := '';
END_VAR
pByte	:= ADR(rValue);

sResult[0]	:= pByte[1];
sResult[1]	:= pByte[0];
sResult[2]	:= pByte[3];
sResult[3]	:= pByte[2];

M_ByteSwap_REAL_TO_STRING	:= sResult;
END_METHOD

METHOD M_ByteSwap_UINT_TO_BYTES : ARRAY [0..1] OF BYTE
VAR_INPUT
	nValue:	UINT;
END_VAR
VAR
	pByte:		POINTER TO BYTE;	// Pointer to nValue
	sResult:	ARRAY [0..1] OF BYTE;
END_VAR
pByte	:= ADR(nValue);

sResult[0]	:= pByte[1];
sResult[1]	:= pByte[0];

M_ByteSwap_UINT_TO_BYTES	:= sResult;
END_METHOD

METHOD M_ByteSwapINT : INT
VAR_INPUT
	pByte:		POINTER TO BYTE;	// Pointer to array of bytes read from JUMO
END_VAR
VAR
	nResult:	INT;
	pResult:	POINTER TO BYTE	:= ADR(nResult);	// Pointer to the result
END_VAR
pResult[0]	:= pByte[1];
pResult[1]	:= pByte[0];

M_ByteSwapINT	:= nResult;
END_METHOD

METHOD M_ByteSwapREAL : REAL
VAR_INPUT
	pByte:		POINTER TO BYTE;	// Pointer to array of bytes read from JUMO
END_VAR
VAR
	rResult:	REAL;
	pResult:	POINTER TO BYTE	:= ADR(rResult);	// Pointer to the result
END_VAR
pResult[0]	:= pByte[1];
pResult[1]	:= pByte[0];
pResult[2]	:= pByte[3];
pResult[3]	:= pByte[2];

M_ByteSwapREAL	:= rResult;
END_METHOD

// Get random value in_lrValue + (in_lrNominator * DRAND)
METHOD M_GenerateRandom_INT : INT
VAR_INPUT
	{attribute 'OPC.UA.DA' := '0'}
	in_lrValue:		LREAL;
	{attribute 'OPC.UA.DA' := '0'}
	in_lrNominator:	LREAL;
END_VAR
VAR
	nVal:	INT;
	lrRand:	LREAL;
	fbDrand:	Tc2_System.DRAND;
END_VAR
VAR_INST
	{attribute 'OPC.UA.DA' := '0'}
	nSeed:	INT := 0;
END_VAR
fbDrand(Seed:=nSeed);
nSeed	:= nSeed + 1;
lrRand	:= in_lrNominator * fbDrand.Num;
nVal	:= LREAL_TO_INT(in_lrValue - in_lrNominator/2.0 + lrRand);

M_GenerateRandom_INT	:= nVal;
END_METHOD

// Get random value in_lrValue + (in_lrNominator * DRAND)
METHOD M_GenerateRandom_REAL : REAL
VAR_INPUT
	{attribute 'OPC.UA.DA' := '0'}
	in_lrValue:		REAL;
	{attribute 'OPC.UA.DA' := '0'}
	in_lrNominator:	REAL;
END_VAR
VAR
	lrVal:	REAL;
	lrRand:	REAL;
	fbDrand:	Tc2_System.DRAND;
END_VAR
VAR_INST
	{attribute 'OPC.UA.DA' := '0'}
	nSeed:	INT := 0;
END_VAR
fbDrand(Seed:=nSeed);
nSeed	:= nSeed + 1;
lrRand	:= LREAL_TO_REAL(in_lrNominator * fbDrand.Num);
lrVal	:= in_lrValue - in_lrNominator/2 + lrRand;	// +- variation

M_GenerateRandom_REAL	:= lrVal;
END_METHOD

METHOD M_GetSimReply : STRING(255)
VAR_INPUT
	{attribute 'OPC.UA.DA' := '0'}
	cmd:	STRING(16);		// MODBUS command. Only first 8 bytes are used
END_VAR
VAR
END_VAR
// TODO User: Implement simulator replies in FBs that EXTEND FB_SIM_MODBUS_COMM_BASE.
//            Only case where cmd[1] = E_MODBUS_CMD_TYPE.READ should be implemented.

IF cmd[1] = E_MODBUS_CMD_TYPE.WRITE THEN
	M_GetSimReply := cmd;	// Reply is the same as the command
ELSE
	M_GetSimReply := '        ';	// Dummy implementation
END_IF
END_METHOD

METHOD M_InsertBytes_INT
VAR_IN_OUT
	s1:	ARRAY [0..300] OF BYTE;;
END_VAR
VAR_INPUT
	s2:	ARRAY [0..1] OF BYTE;;
	nPos:	INT;
END_VAR
VAR
	i:	INT;
END_VAR
FOR i:= 0 TO 1 DO
	s1[nPos+i]	:= s2[i];
END_FOR
END_METHOD

METHOD M_InsertBytes_REAL
VAR_IN_OUT
	s1:	ARRAY [0..300] OF BYTE;;
END_VAR
VAR_INPUT
	s2:	ARRAY [0..3] OF BYTE;;
	nPos:	INT;
END_VAR
VAR
	i:	INT;
END_VAR
FOR i:= 0 TO 3 DO
	s1[nPos+i]	:= s2[i];
END_FOR
END_METHOD

END_FUNCTION_BLOCK

// POUs/FB_SIM_MODBUS_COMM_JUMO
FUNCTION_BLOCK FB_SIM_MODBUS_COMM_JUMO EXTENDS FB_SIM_MODBUS_COMM_BASE
VAR_INPUT
END_VAR
VAR_OUTPUT
END_VAR
VAR
END_VAR

M_ActivityDo();

METHOD M_GetSimReply : STRING(255)
VAR_INPUT
	{attribute 'OPC.UA.DA' := '0'}
	cmd:	STRING(16);		// MODBUS command. Only first 8 bytes are used
END_VAR
VAR
	sReply:	STRING(255);
	sTmp:	STRING(8);
	i,j:	INT;
	pByte:	POINTER TO BYTE;
	rReal:	REAL;
	nRegister:	INT;
	nWords:	INT;	
END_VAR
// TODO User: Implement simulator replies in FBs that EXTEND FB_SIM_MODBUS_COMM_BASE.
//            Only case where cmd[1] = E_MODBUS_CMD_TYPE.READ should be implemented.

IF cmd[1] = E_MODBUS_CMD_TYPE.WRITE THEN
	M_GetSimReply := cmd;	// Reply is the same as the command
ELSE
	// Get register number - cmd[2..3] swapped bytes
	nRegister	:= M_ByteSwapINT(ADR(cmd[2]));

	// Get number of words - cmd[4..5] swapped bytes
	nWords	:= M_ByteSwapINT(ADR(cmd[4]));

	sReply[0]	:= cmd[0];
	sReply[1]	:= cmd[1];
	sReply[2]	:= INT_TO_BYTE(nWords * 2);
	
	IF nRegister = 16#00A4 THEN		// common data
		FOR i := 1 TO 54 DO
			sTmp := M_ByteSwap_REAL_TO_STRING(M_GenerateRandom_REAL(100.0,10));
			FOR j := 0 TO 3 DO
				sReply[3 + (i-1)*4 + j]	:= sTmp[j];
			END_FOR
		END_FOR
		// - Switch Stats, offset 3 + 54x4 = 219 (111 is not correct!!!)
		FOR i := 1 TO 8 DO
			sTmp := M_ByteSwap_INT_TO_STRING(M_GenerateRandom_INT(0.5,1.0));
			FOR j := 0 TO 1 DO
				sReply[111 + (i-1)*2 + j]	:= sTmp[j];
			END_FOR
		END_FOR
	ELSIF nRegister = 16#083C THEN	// set points
		FOR i := 1 TO 16 DO
			sTmp := M_ByteSwap_REAL_TO_STRING(M_GenerateRandom_REAL(80.0,1.0));
			FOR j := 0 TO 3 DO
				sReply[3 + (i-1)*4 + j]	:= sTmp[j];
			END_FOR
		END_FOR
	END_IF
	
	// TODO
	// Calculate CRC for the first 6 bytes
	//	crc	:= M_CRC(ADR(cmd),6);
	

	M_GetSimReply := sReply;
END_IF
END_METHOD

END_FUNCTION_BLOCK

// POUs/FB_SIM_RS_COMM_BASE
FUNCTION_BLOCK FB_SIM_RS_COMM_BASE
VAR_INPUT
	in_nModel:			DINT;
	in_sReplySuffix:	STRING(16);	// Terminator for reply
END_VAR
VAR_OUTPUT
END_VAR
VAR
END_VAR

M_ActivityDo();

METHOD M_ActivityDo
VAR_INPUT
END_VAR
END_METHOD

// Get random value in_lrValue + (in_lrNominator * DRAND)
METHOD M_GenerateRandom_LREAL : LREAL
VAR_INPUT
	{attribute 'OPC.UA.DA' := '0'}
	in_lrValue:		LREAL;
	{attribute 'OPC.UA.DA' := '0'}
	in_lrNominator:	LREAL;
END_VAR
VAR
	lrVal:	LREAL;
	lrRand:	LREAL;
	fbDrand:	Tc2_System.DRAND;
END_VAR
VAR_INST
	{attribute 'OPC.UA.DA' := '0'}
	nSeed:	INT := 0;
END_VAR
fbDrand(Seed:=nSeed);
nSeed	:= nSeed + 1;
lrRand	:= in_lrNominator * fbDrand.Num;
lrVal	:= in_lrValue + lrRand;

M_GenerateRandom_LREAL	:= lrVal;
END_METHOD

// Get string with terminator. 
METHOD M_Get_INT_TO_STRING : STRING(255)
VAR_INPUT
	{attribute 'OPC.UA.DA' := '0'}
	in_nValue:		INT;
END_VAR
VAR
END_VAR
// Add sufix, if any
IF in_sReplySuffix <> '' THEN
	M_Get_INT_TO_STRING	:= CONCAT (INT_TO_STRING(in_nValue),in_sReplySuffix);
ELSE
	M_Get_INT_TO_STRING	:= INT_TO_STRING(in_nValue);
END_IF
END_METHOD

// Get string with given precision and add terminator. 
METHOD M_Get_LREAL_TO_STRING : STRING(255)
VAR_INPUT
	{attribute 'OPC.UA.DA' := '0'}
	in_lrValue:		LREAL;
	{attribute 'OPC.UA.DA' := '0'}
	in_nPrecision:	INT	:= 2;	// Number of decimal places, default 2
END_VAR
VAR
	lrVal:		LREAL;
    fbFormat:	FB_FormatString;
	sFormat:	STRING;
    sVal:		T_MaxString;
END_VAR
// Get the input value
lrVal	:= in_lrValue;
// Create a string like '%.2f'
sFormat	:= CONCAT(CONCAT('%.', INT_TO_STRING(in_nPrecision)),'f');
// Print LREAL with <in_nPrecision> decimal places
fbFormat( sFormat := sFormat, arg1 := F_LREAL( lrVal ), sOut => sVal);

// Add sufix, if any
IF in_sReplySuffix <> '' THEN
	M_Get_LREAL_TO_STRING	:= CONCAT (sVal,in_sReplySuffix);
ELSE
	M_Get_LREAL_TO_STRING	:= sVal;
END_IF
END_METHOD

METHOD M_GetRandom_LREAL_TO_STRING : STRING(255)
VAR_INPUT
	{attribute 'OPC.UA.DA' := '0'}
	in_lrValue:		LREAL;
	{attribute 'OPC.UA.DA' := '0'}
	in_lrNominator:	LREAL;
	{attribute 'OPC.UA.DA' := '0'}
	in_nPrecision:	INT	:= 2;	// Number of decimal places, default 2
END_VAR
VAR
	lrVal:		LREAL;
    fbFormat:	FB_FormatString;
	sFormat:	STRING;
    sVal:		T_MaxString;
END_VAR
// Get a random value
lrVal	:= M_GenerateRandom_LREAL(in_lrValue,in_lrNominator);
// Create a string like '%.2f'
sFormat	:= CONCAT(CONCAT('%.', INT_TO_STRING(in_nPrecision)),'f');
// Print LREAL with <in_nPrecision> decimal places
fbFormat( sFormat := sFormat, arg1 := F_LREAL( lrVal ), sOut => sVal);

// Add sufix, if any
IF in_sReplySuffix <> '' THEN
	M_GetRandom_LREAL_TO_STRING	:= CONCAT (sVal,in_sReplySuffix);
ELSE
	M_GetRandom_LREAL_TO_STRING	:= sVal;
END_IF
END_METHOD

METHOD M_GetSimReply : STRING(255)
VAR_INPUT
	{attribute 'OPC.UA.DA' := '0'}
	in_sReceived:	STRING(255);		// String received from a client
END_VAR
VAR
END_VAR
// TODO User: Implement simulater replies in FBs that EXTEND FB_SIM_RS_COMM_BASE.
M_GetSimReply := '';	// Dummy implementation
END_METHOD

END_FUNCTION_BLOCK

// POUs/FB_SIM_RS_COMM_DUMMY
FUNCTION_BLOCK FB_SIM_RS_COMM_DUMMY EXTENDS FB_SIM_RS_COMM_BASE
VAR_INPUT
END_VAR
VAR_OUTPUT
END_VAR
VAR
	//
	// TODO: Status structure for <devices>.
	// See also: FB_SIM_RS_COMM_LAKESHORE.
	//
	
	fbTimer:		TON;	// Used for ramps etc.

END_VAR

M_ActivityDo();	// Implement ramps, etc, if any

METHOD M_ActivityDo
VAR_INPUT
END_VAR
// TODO User: Implement ramps, if any.
END_METHOD

METHOD M_GetSimReply : STRING(255)
VAR_INPUT
	{attribute 'OPC.UA.DA' := '0'}
	in_sReceived:	STRING(255);		// String received from a client
END_VAR
VAR
	sReply:	STRING(255);
	lrVal:	LREAL;
	i:		INT;
    fbFormat   : FB_FormatString;
    sOut       : T_MaxString;
	nCh:	INT := 8;	// Number of channels for models 218 and 224
END_VAR
// TODO User: Implement simulated replies.

// Dummy empty reply
M_GetSimReply	:= in_sReplySuffix;
END_METHOD

END_FUNCTION_BLOCK

// POUs/FB_SIM_RS_COMM_LAKESHORE
FUNCTION_BLOCK FB_SIM_RS_COMM_LAKESHORE EXTENDS FB_SIM_RS_COMM_BASE
VAR_INPUT
END_VAR
VAR_OUTPUT
END_VAR
VAR
	//
	// Status structure for Lakeshore devices
	//
	bRAMP_On:		BOOL	:= FALSE;	// RAMP On/Off state
	nPID_P:			UINT	:= 10;		// PID parameter P
	nPID_I:			UINT	:= 50;		// PID parameter I
	nPID_D:			UINT	:= 40;		// PID parameter D
	lrKRDG_A:		LREAL	:= 283.15;	// Temperature A [K]
	lrKRDG_B:		LREAL	:= 273.15;	// Temperature B [K]
	lrCRDG_A:		LREAL	:= 10.0;	// Temperature A [C]
	lrCRDG_B:		LREAL	:=  0.0;	// Temperature B [C]
	lrRAMP_Rate:	LREAL	:= 0.0;		// RAMP rate
	lrSETP:			LREAL	:= 283.15;	// Actual Setpoint [K]
	lrSETP_Target:	LREAL	:= 283.15;	// Target Setpoint [K]
	lrHTR:			LREAL	:= 0.0;		// Heater output [%]
	nRANGE:			UINT	:= 4;		// Heater range
	
	fbTimer:		TON;

END_VAR

M_ActivityDo();	// Implement ramps, if any

METHOD M_ActivityDo
VAR_INPUT
END_VAR
// TODO User: Implement ramps, if any.
END_METHOD

METHOD M_GetSimReply : STRING(255)
VAR_INPUT
	{attribute 'OPC.UA.DA' := '0'}
	in_sReceived:	STRING(255);		// String received from a client
END_VAR
VAR
	sReply:	STRING(255);
	lrVal:	LREAL;
	i:		INT;
    fbFormat   : FB_FormatString;
    sOut       : T_MaxString;
	nCh:	INT := 8;	// Number of channels for models 218 and 224
END_VAR
IF in_nModel = 340 THEN
	IF FIND (in_sReceived, '*IDN?') > 0 THEN
		M_GetSimReply	:= CONCAT('Lakeshore Simulator',in_sReplySuffix);
	ELSIF FIND (in_sReceived, '*') = 1 THEN
		M_GetSimReply	:= '';	// Ignore commands starting with '*'
	ELSIF FIND (in_sReceived, 'MODE ') > 0 THEN
		M_GetSimReply	:= '';
	ELSIF FIND (in_sReceived, 'CRDG? A') > 0 THEN
		M_GetSimReply	:= M_GetRandom_LREAL_TO_STRING(lrCRDG_A,0.01,2);
	ELSIF FIND (in_sReceived, 'KRDG? A') > 0 THEN
		M_GetSimReply	:= M_GetRandom_LREAL_TO_STRING(lrKRDG_A,0.01,2);
	ELSIF FIND (in_sReceived, 'CRDG? B') > 0 THEN
		M_GetSimReply	:= M_GetRandom_LREAL_TO_STRING(lrCRDG_B,0.01,2);
	ELSIF FIND (in_sReceived, 'KRDG? B') > 0 THEN
		M_GetSimReply	:= M_GetRandom_LREAL_TO_STRING(lrKRDG_B,0.01,2);
	ELSIF FIND (in_sReceived, 'SETP?') > 0 THEN
		M_GetSimReply	:= M_Get_LREAL_TO_STRING(lrSETP_Target,2);
	ELSIF FIND (in_sReceived, 'PID?') > 0 THEN
		fbFormat(	sFormat := '%d,%d,%d', 
					arg1 := F_UINT(nPID_P), 
					arg2 := F_UINT(nPID_I), 
					arg3 := F_UINT(nPID_D), 
					sOut => sOut);
		M_GetSimReply	:= CONCAT(sOut,in_sReplySuffix);
	ELSIF FIND (in_sReceived, 'RANGE?') > 0 THEN
		M_GetSimReply	:= M_Get_INT_TO_STRING(UINT_TO_INT(nRANGE));
	ELSIF FIND (in_sReceived, 'HTR?') > 0 THEN
		M_GetSimReply	:= M_GetRandom_LREAL_TO_STRING(lrHTR,0.10,2);
	ELSIF FIND (in_sReceived, 'AOUT?') > 0 THEN
		M_GetSimReply	:= M_GetRandom_LREAL_TO_STRING(0.0,0.10,2);
	ELSE
		M_GetSimReply	:= CONCAT('777.77',in_sReplySuffix);
	END_IF
ELSIF in_nModel = 336 THEN
	IF FIND (in_sReceived, 'MODE 1') > 0 THEN
		M_GetSimReply	:= '';
	ELSIF FIND (in_sReceived, '*IDN?') > 0 THEN
		M_GetSimReply	:= CONCAT('Lakeshore Simulator',in_sReplySuffix);
	ELSIF FIND (in_sReceived, 'CRDG?') > 0 THEN
		M_GetSimReply	:= M_GetRandom_LREAL_TO_STRING(-233.15,0.10,2);
	ELSIF FIND (in_sReceived, 'KRDG?') > 0 THEN
		M_GetSimReply	:= M_GetRandom_LREAL_TO_STRING(40,0.10,2);
	ELSIF FIND (in_sReceived, 'SETP?') > 0 THEN
		M_GetSimReply	:= '40.00$0D$0A';
	ELSIF FIND (in_sReceived, 'PID?') > 0 THEN
		fbFormat(	sFormat := '%d,%d,%d', 
					arg1 := F_UINT(nPID_P), 
					arg2 := F_UINT(nPID_I), 
					arg3 := F_UINT(nPID_D), sOut => sOut);
		M_GetSimReply	:= CONCAT(sOut,in_sReplySuffix);
	ELSIF FIND (in_sReceived, 'RANGE?') > 0 THEN
		M_GetSimReply	:= '1$0D$0A';
	ELSIF FIND (in_sReceived, 'HTR?') > 0 THEN
		M_GetSimReply	:= M_GetRandom_LREAL_TO_STRING(25,0.10,2);
	ELSIF FIND (in_sReceived, 'AOUT?') > 0 THEN
		M_GetSimReply	:= M_GetRandom_LREAL_TO_STRING(45,0.10,2);
	ELSE
		M_GetSimReply	:= CONCAT('777.77',in_sReplySuffix);
	END_IF
ELSIF in_nModel = 218  OR  in_nModel = 224 THEN
	IF in_nModel = 218 THEN
		nCh	:= 8;
	ELSIF in_nModel = 224 THEN
		nCh	:= 12;
	END_IF
	IF FIND (in_sReceived, 'MODE 1') > 0 THEN
		M_GetSimReply	:= '';
	ELSIF FIND (in_sReceived, '*IDN?') > 0 THEN
		M_GetSimReply	:= CONCAT('Lakeshore Simulator',in_sReplySuffix);
	ELSIF FIND (in_sReceived, 'CRDG?') > 0 THEN
		// Generate a string like:
		// '-233.15,-233.25,-233.35,-233.45,-233.55,-233.65,-233.75,-233.85,-233.95,-233.15,-233.25,-233.35$0D$0A';
		sReply	:= '';
		FOR i:=1 TO nCh DO
			lrVal	:= M_GenerateRandom_LREAL(lrCRDG_A,0.10);
			IF i < nCh THEN
				fbFormat( sFormat := '%+.2f,', arg1 := F_LREAL( lrVal ), sOut => sOut);
			ELSE				
				fbFormat( sFormat := '%+.2f%s', arg1 := F_LREAL( lrVal ), arg2 := F_STRING( in_sReceived ), sOut => sOut);
			END_IF
			sReply	:= CONCAT(sReply, sOut);
		END_FOR
		M_GetSimReply	:= sReply;
	ELSIF FIND (in_sReceived, 'KRDG?') > 0 THEN
		// Generate a string like:
		// '40.15,40.25,40.35,40.45,40.55,40.65,40.75,40.85,40.95,40.15,40.25,40.35$0D$0A';
		sReply	:= '';
		FOR i:=1 TO nCh DO
			lrVal	:= M_GenerateRandom_LREAL(lrKRDG_A,0.10);
			IF i < nCh THEN
				fbFormat( sFormat := '%+.2f,', arg1 := F_LREAL( lrVal ), sOut => sOut);
			ELSE				
				fbFormat( sFormat := '%+.2f%s', arg1 := F_LREAL( lrVal ), arg2 := F_STRING( in_sReceived ), sOut => sOut);
			END_IF
			sReply	:= CONCAT(sReply, sOut);
		END_FOR
		M_GetSimReply	:= sReply;
	ELSE
		M_GetSimReply	:= CONCAT('777.77',in_sReplySuffix);
	END_IF
END_IF
END_METHOD

END_FUNCTION_BLOCK

// POUs/MAIN
PROGRAM MAIN
VAR
END_VAR

END_PROGRAM
